// TwinCAT 3 PLC project ExternControl
// ProgramVersion: 3.1.4026.19
// libraries:
//   Tc2_Standard, * (Beckhoff Automation GmbH)
//   Tc2_System, * (Beckhoff Automation GmbH)
//   Tc2_Utilities, * (Beckhoff Automation GmbH)
//   VisuDialogs, * (System)
//   VisuDialogs
// project tree:
//   APPLICATION/ fb_Simulation.TcPOU, GVL_APPLICATION.TcGVL, MAIN_APP.TcPOU
//   APPLICATION/_types/ E_PROCESS_CHECK.TcDUT (not stored), E_PROCESS_CTRL.TcDUT (not stored), E_PROCESS_STATE.TcDUT (not stored), ST_PROCESS_CTRL.TcDUT (not stored), ST_PROCESS_STATE.TcDUT (not stored), T_PROCESS.TcDUT (not stored)
//   APPLICATION/_types/fb_Instance/ E_INSTANCE_CHECK.TcDUT, E_INSTANCE_STATE.TcDUT (not stored), fb_Instance.TcPOU (not stored)
//   APPLICATION/_types/LinkedList/ fb_Process_LinkedListCtrl.TcPOU (not stored), I_Process_LinkedList.TcIO (not stored), ST_PROCESS_DATA.TcDUT (not stored), ST_PROCESS_LIST_RESULT.TcDUT (not stored)
//   / GlobalTextList.TcGTLO (not stored), MAIN.TcPOU (not stored), PlcTask.TcTTO, Visualization Manager.TcVMO (not stored)
//   MAPPING/ MAPPING_in.TcPOU (not stored), MAPPING_out.TcPOU (not stored)
//   MAPPING/_types/ U_APP_CTRL.TcDUT (not stored), U_APP_STATE.TcDUT (not stored), U_INSTANCE_CTRL.TcDUT (not stored), U_INSTANCE_STATE.TcDUT (not stored), U_TICKET_LIST_CTRL.TcDUT (not stored), U_TICKET_LIST_DATA_INPUT.TcDUT (not stored), U_TICKET_LIST_DATA_OUTPUT.TcDUT (not stored), U_TICKET_LIST_STATE.TcDUT (not stored), U_XTS_STATION_CTRL.TcDUT (not stored), U_XTS_STATION_STATE.TcDUT (not stored), U_XTS_TRANSPORT_CTRL.TcDUT, U_XTS_TRANSPORT_STATE.TcDUT (not stored)
//   MSG/ fb_LocalTime.TcPOU (not stored), fb_MessageData.TcPOU (not stored), fb_MessageDataCtrl.TcPOU, f_MessageSet.TcPOU (not stored), GVL_MSG.TcGVL (not stored), I_MessageData.TcIO
//   MSG/types/ e_Device.TcDUT (not stored), E_MessageType.TcDUT (not stored), E_MESSAGE_BATCH.TcDUT (not stored), E_MESSAGE_CHECK.TcDUT (not stored), E_MESSAGE_CTRL.TcDUT (not stored), E_MESSAGE_FLOW.TcDUT (not stored), E_MESSAGE_STATE.TcDUT, e_Subdevice.TcDUT (not stored), ST_Message.TcDUT (not stored), ST_MESSAGE_CTRL.TcDUT (not stored), ST_MESSAGE_STATE.TcDUT (not stored), TL_E_MESSAGETYPE.TcTLO
//   XTS/CaGroup/types/ E_CA_GROUP_STATE.TcDUT (not stored), E_GROUP_CHECK.TcDUT (not stored), ST_GROUP_INFO.TcDUT
//   XTS/ GVL_XTS.TcGVL (not stored), XTS_Parameter.TcGVL (not stored)
//   XTS/Mover/types/ E_MOVER_CTRL.TcDUT (not stored), E_MOVER_STATE.TcDUT (not stored), ST_GEAR_DATA.TcDUT (not stored), ST_MOVER_CTRL.TcDUT (not stored), ST_MOVER_INFO.TcDUT, ST_MOVER_STATE.TcDUT (not stored), ST_MOVE_DATA.TcDUT (not stored)
//   XTS/Xpu/types/ E_XPU_CHECK.TcDUT (not stored), E_XPU_CTRL.TcDUT (not stored), E_XPU_INIT.TcDUT (not stored), E_XPU_STATE.TcDUT (not stored), ST_XPU_CTRL.TcDUT (not stored), ST_XPU_INFO.TcDUT, ST_XPU_STATE.TcDUT (not stored)
//   XTS/XtsStation/_types/ E_STATION_CTRL.TcDUT (not stored), E_STATION_GEAR_DISTANCE_AXIS.TcDUT (not stored), E_STATION_STATE.TcDUT (not stored), E_STATION_TYPE.TcDUT (not stored), ST_STATION_CTRL.TcDUT (not stored), ST_STATION_GEAR_PARAMETER.TcDUT (not stored), ST_STATION_LIST_RESULT.TcDUT (not stored), ST_STATION_MOVER_DATA.TcDUT (not stored), ST_STATION_PARAMETER.TcDUT, ST_STATION_STATE.TcDUT (not stored), T_NEST_OFFSET.TcDUT
//   XTS/XtsTransportUnit/types/ E_XTS_TRANSPORT_CHECK.TcDUT (not stored), E_XTS_TRANSPORT_CTRL.TcDUT (not stored), E_XTS_TRANSPORT_STATE.TcDUT (not stored), ST_XTS_TRANSPORT_CTRL.TcDUT (not stored), ST_XTS_TRANSPORT_STATE.TcDUT (not stored)
//   XTS/_types/ E_PROGRESS.TcDUT (not stored), f_GetProgress.TcPOU (not stored), f_GetState.TcPOU (not stored)
//   XTS/_Visualization/ GROUP_VISU.TcVIS (not stored), MOVER_VISU.TcVIS (not stored), STATION_VISU.TcVIS (not stored), XPU_VISU.TcVIS (not stored), XTS_TRANSPORT.TcVIS (not stored)
//   XTS/_Visualization/textlists/ TL_E_CTRL_MOVER.TcTLO (not stored), TL_E_CTRL_STATION.TcTLO (not stored), TL_E_CTRL_TRANSPORT.TcTLO (not stored), TL_E_CTRL_XPU.TcTLO (not stored)
//   XTS/_Visualization/types/ ST_XPU_STRINGS.TcDUT (not stored)
// real-time tasks:
//   TASK XTS Task 1: cycle T#250us, priority 1, ADS port 350
//   TASK XTS AUX Task 1: cycle T#250us, priority 2, ADS port 351
//   TASK XTS Task 2: cycle T#250us, priority 3, ADS port 352
//   TASK PlcTask: cycle T#2ms, priority 15, ADS port 353
//   TASK Job Task: cycle default, priority 32
// motion (NC):
//   TASK NC-Task 1: cycle T#2ms, priority 4, ADS port 501
//   TASK NC-Task 1 SVB: cycle T#10ms, priority 8, ADS port 511
//   AXIS Mover Axis 1 (id 1)
//     Dynamic: AccelerationMaximum=80000, DecelerationMaximum=80000, Acceleration=20000, Deceleration=20000, Jerk=200000
//     Velo: Maximum=4000
//     PositionAreaControl: Enable=false
//     TargetPosControl: Enable=false
//     OtherSettings: AllowMotionCmdToSlave=true, AllowMotionCmdToExtSetGenAxis=true
//     encoder EncType=28
//       EncPara: ModuloFactor=8000, ToleranceWndModuloStart=0.2, MaxCount=#xffffffff
//     drive DrvType=22
//       DrvPara: MaxCount=#xffffffff, DriveControlDWord=#x00000100
//         Analog: VeloReferenz=4200, TorqueSetpointScale=10
//         TimeComp: TaskDelayCycles=1
//     controller CtrType=1
//       CtrPara: PriorControlFactor=1
//         PosDiffControl: Range=10
//         Observer: BandWidth=20
//   AXIS Mover Axis 2 (id 2)
//     Dynamic: AccelerationMaximum=80000, DecelerationMaximum=80000, Acceleration=20000, Deceleration=20000, Jerk=200000
//     Velo: Maximum=4000
//     PositionAreaControl: Enable=false
//     TargetPosControl: Enable=false
//     OtherSettings: AllowMotionCmdToSlave=true, AllowMotionCmdToExtSetGenAxis=true
//     encoder EncType=28
//       EncPara: ModuloFactor=8000, ToleranceWndModuloStart=0.2, MaxCount=#xffffffff
//     drive DrvType=22
//       DrvPara: MaxCount=#xffffffff, DriveControlDWord=#x00000100
//         Analog: VeloReferenz=4200, TorqueSetpointScale=10
//         TimeComp: TaskDelayCycles=1
//     controller CtrType=1
//       CtrPara: PriorControlFactor=1
//         PosDiffControl: Range=10
//         Observer: BandWidth=20
//   AXIS Mover Axis 3 (id 3)
//     Dynamic: AccelerationMaximum=80000, DecelerationMaximum=80000, Acceleration=20000, Deceleration=20000, Jerk=200000
//     Velo: Maximum=4000
//     PositionAreaControl: Enable=false
//     TargetPosControl: Enable=false
//     OtherSettings: AllowMotionCmdToSlave=true, AllowMotionCmdToExtSetGenAxis=true
//     encoder EncType=28
//       EncPara: ModuloFactor=8000, ToleranceWndModuloStart=0.2, MaxCount=#xffffffff
//     drive DrvType=22
//       DrvPara: MaxCount=#xffffffff, DriveControlDWord=#x00000100
//         Analog: VeloReferenz=4200, TorqueSetpointScale=10
//         TimeComp: TaskDelayCycles=1
//     controller CtrType=1
//       CtrPara: PriorControlFactor=1
//         PosDiffControl: Range=10
//         Observer: BandWidth=20
//   AXIS Mover Axis 4 (id 4)
//     Dynamic: AccelerationMaximum=80000, DecelerationMaximum=80000, Acceleration=20000, Deceleration=20000, Jerk=200000
//     Velo: Maximum=4000
//     PositionAreaControl: Enable=false
//     TargetPosControl: Enable=false
//     OtherSettings: AllowMotionCmdToSlave=true, AllowMotionCmdToExtSetGenAxis=true
//     encoder EncType=28
//       EncPara: ModuloFactor=8000, ToleranceWndModuloStart=0.2, MaxCount=#xffffffff
//     drive DrvType=22
//       DrvPara: MaxCount=#xffffffff, DriveControlDWord=#x00000100
//         Analog: VeloReferenz=4200, TorqueSetpointScale=10
//         TimeComp: TaskDelayCycles=1
//     controller CtrType=1
//       CtrPara: PriorControlFactor=1
//         PosDiffControl: Range=10
//         Observer: BandWidth=20
//   AXIS Mover Axis 5 (id 5)
//     Dynamic: AccelerationMaximum=80000, DecelerationMaximum=80000, Acceleration=20000, Deceleration=20000, Jerk=200000
//     Velo: Maximum=4000
//     PositionAreaControl: Enable=false
//     TargetPosControl: Enable=false
//     OtherSettings: AllowMotionCmdToSlave=true, AllowMotionCmdToExtSetGenAxis=true
//     encoder EncType=28
//       EncPara: ModuloFactor=8000, ToleranceWndModuloStart=0.2, MaxCount=#xffffffff
//     drive DrvType=22
//       DrvPara: MaxCount=#xffffffff, DriveControlDWord=#x00000100
//         Analog: VeloReferenz=4200, TorqueSetpointScale=10
//         TimeComp: TaskDelayCycles=1
//     controller CtrType=1
//       CtrPara: PriorControlFactor=1
//         PosDiffControl: Range=10
//         Observer: BandWidth=20
//   AXIS Mover Axis 6 (id 6)
//     Dynamic: AccelerationMaximum=80000, DecelerationMaximum=80000, Acceleration=20000, Deceleration=20000, Jerk=200000
//     Velo: Maximum=4000
//     PositionAreaControl: Enable=false
//     TargetPosControl: Enable=false
//     OtherSettings: AllowMotionCmdToSlave=true, AllowMotionCmdToExtSetGenAxis=true
//     encoder EncType=28
//       EncPara: ModuloFactor=8000, ToleranceWndModuloStart=0.2, MaxCount=#xffffffff
//     drive DrvType=22
//       DrvPara: MaxCount=#xffffffff, DriveControlDWord=#x00000100
//         Analog: VeloReferenz=4200, TorqueSetpointScale=10
//         TimeComp: TaskDelayCycles=1
//     controller CtrType=1
//       CtrPara: PriorControlFactor=1
//         PosDiffControl: Range=10
//         Observer: BandWidth=20
//   AXIS Mover Axis 7 (id 7)
//     Dynamic: AccelerationMaximum=80000, DecelerationMaximum=80000, Acceleration=20000, Deceleration=20000, Jerk=200000
//     Velo: Maximum=4000
//     PositionAreaControl: Enable=false
//     TargetPosControl: Enable=false
//     OtherSettings: AllowMotionCmdToSlave=true, AllowMotionCmdToExtSetGenAxis=true
//     encoder EncType=28
//       EncPara: ModuloFactor=8000, ToleranceWndModuloStart=0.2, MaxCount=#xffffffff
//     drive DrvType=22
//       DrvPara: MaxCount=#xffffffff, DriveControlDWord=#x00000100
//         Analog: VeloReferenz=4200, TorqueSetpointScale=10
//         TimeComp: TaskDelayCycles=1
//     controller CtrType=1
//       CtrPara: PriorControlFactor=1
//         PosDiffControl: Range=10
//         Observer: BandWidth=20
//   AXIS Mover Axis 8 (id 8)
//     Dynamic: AccelerationMaximum=80000, DecelerationMaximum=80000, Acceleration=20000, Deceleration=20000, Jerk=200000
//     Velo: Maximum=4000
//     PositionAreaControl: Enable=false
//     TargetPosControl: Enable=false
//     OtherSettings: AllowMotionCmdToSlave=true, AllowMotionCmdToExtSetGenAxis=true
//     encoder EncType=28
//       EncPara: ModuloFactor=8000, ToleranceWndModuloStart=0.2, MaxCount=#xffffffff
//     drive DrvType=22
//       DrvPara: MaxCount=#xffffffff, DriveControlDWord=#x00000100
//         Analog: VeloReferenz=4200, TorqueSetpointScale=10
//         TimeComp: TaskDelayCycles=1
//     controller CtrType=1
//       CtrPara: PriorControlFactor=1
//         PosDiffControl: Range=10
//         Observer: BandWidth=20
//   AXIS Mover Axis 9 (id 9)
//     Dynamic: AccelerationMaximum=80000, DecelerationMaximum=80000, Acceleration=20000, Deceleration=20000, Jerk=200000
//     Velo: Maximum=4000
//     PositionAreaControl: Enable=false
//     TargetPosControl: Enable=false
//     OtherSettings: AllowMotionCmdToSlave=true, AllowMotionCmdToExtSetGenAxis=true
//     encoder EncType=28
//       EncPara: ModuloFactor=8000, ToleranceWndModuloStart=0.2, MaxCount=#xffffffff
//     drive DrvType=22
//       DrvPara: MaxCount=#xffffffff, DriveControlDWord=#x00000100
//         Analog: VeloReferenz=4200, TorqueSetpointScale=10
//         TimeComp: TaskDelayCycles=1
//     controller CtrType=1
//       CtrPara: PriorControlFactor=1
//         PosDiffControl: Range=10
//         Observer: BandWidth=20
//   AXIS Mover Axis 10 (id 10)
//     Dynamic: AccelerationMaximum=80000, DecelerationMaximum=80000, Acceleration=20000, Deceleration=20000, Jerk=200000
//     Velo: Maximum=4000
//     PositionAreaControl: Enable=false
//     TargetPosControl: Enable=false
//     OtherSettings: AllowMotionCmdToSlave=true, AllowMotionCmdToExtSetGenAxis=true
//     encoder EncType=28
//       EncPara: ModuloFactor=8000, ToleranceWndModuloStart=0.2, MaxCount=#xffffffff
//     drive DrvType=22
//       DrvPara: MaxCount=#xffffffff, DriveControlDWord=#x00000100
//         Analog: VeloReferenz=4200, TorqueSetpointScale=10
//         TimeComp: TaskDelayCycles=1
//     controller CtrType=1
//       CtrPara: PriorControlFactor=1
//         PosDiffControl: Range=10
//         Observer: BandWidth=20
//   AXIS Mover Axis 11 (id 11)
//     Dynamic: AccelerationMaximum=80000, DecelerationMaximum=80000, Acceleration=20000, Deceleration=20000, Jerk=200000
//     Velo: Maximum=4000
//     PositionAreaControl: Enable=false
//     TargetPosControl: Enable=false
//     OtherSettings: AllowMotionCmdToSlave=true, AllowMotionCmdToExtSetGenAxis=true
//     encoder EncType=28
//       EncPara: ModuloFactor=8000, ToleranceWndModuloStart=0.2, MaxCount=#xffffffff
//     drive DrvType=22
//       DrvPara: MaxCount=#xffffffff, DriveControlDWord=#x00000100
//         Analog: VeloReferenz=4200, TorqueSetpointScale=10
//         TimeComp: TaskDelayCycles=1
//     controller CtrType=1
//       CtrPara: PriorControlFactor=1
//         PosDiffControl: Range=10
//         Observer: BandWidth=20
//   AXIS Mover Axis 12 (id 12)
//     Dynamic: AccelerationMaximum=80000, DecelerationMaximum=80000, Acceleration=20000, Deceleration=20000, Jerk=200000
//     Velo: Maximum=4000
//     PositionAreaControl: Enable=false
//     TargetPosControl: Enable=false
//     OtherSettings: AllowMotionCmdToSlave=true, AllowMotionCmdToExtSetGenAxis=true
//     encoder EncType=28
//       EncPara: ModuloFactor=8000, ToleranceWndModuloStart=0.2, MaxCount=#xffffffff
//     drive DrvType=22
//       DrvPara: MaxCount=#xffffffff, DriveControlDWord=#x00000100
//         Analog: VeloReferenz=4200, TorqueSetpointScale=10
//         TimeComp: TaskDelayCycles=1
//     controller CtrType=1
//       CtrPara: PriorControlFactor=1
//         PosDiffControl: Range=10
//         Observer: BandWidth=20
//   AXIS Mover Axis 13 (id 13)
//     Dynamic: AccelerationMaximum=80000, DecelerationMaximum=80000, Acceleration=20000, Deceleration=20000, Jerk=200000
//     Velo: Maximum=4000
//     PositionAreaControl: Enable=false
//     TargetPosControl: Enable=false
//     OtherSettings: AllowMotionCmdToSlave=true, AllowMotionCmdToExtSetGenAxis=true
//     encoder EncType=28
//       EncPara: ModuloFactor=8000, ToleranceWndModuloStart=0.2, MaxCount=#xffffffff
//     drive DrvType=22
//       DrvPara: MaxCount=#xffffffff, DriveControlDWord=#x00000100
//         Analog: VeloReferenz=4200, TorqueSetpointScale=10
//         TimeComp: TaskDelayCycles=1
//     controller CtrType=1
//       CtrPara: PriorControlFactor=1
//         PosDiffControl: Range=10
//         Observer: BandWidth=20
//   AXIS Mover Axis 14 (id 14)
//     Dynamic: AccelerationMaximum=80000, DecelerationMaximum=80000, Acceleration=20000, Deceleration=20000, Jerk=200000
//     Velo: Maximum=4000
//     PositionAreaControl: Enable=false
//     TargetPosControl: Enable=false
//     OtherSettings: AllowMotionCmdToSlave=true, AllowMotionCmdToExtSetGenAxis=true
//     encoder EncType=28
//       EncPara: ModuloFactor=8000, ToleranceWndModuloStart=0.2, MaxCount=#xffffffff
//     drive DrvType=22
//       DrvPara: MaxCount=#xffffffff, DriveControlDWord=#x00000100
//         Analog: VeloReferenz=4200, TorqueSetpointScale=10
//         TimeComp: TaskDelayCycles=1
//     controller CtrType=1
//       CtrPara: PriorControlFactor=1
//         PosDiffControl: Range=10
//         Observer: BandWidth=20
//   AXIS Mover Axis 15 (id 15)
//     Dynamic: AccelerationMaximum=80000, DecelerationMaximum=80000, Acceleration=20000, Deceleration=20000, Jerk=200000
//     Velo: Maximum=4000
//     PositionAreaControl: Enable=false
//     TargetPosControl: Enable=false
//     OtherSettings: AllowMotionCmdToSlave=true, AllowMotionCmdToExtSetGenAxis=true
//     encoder EncType=28
//       EncPara: ModuloFactor=8000, ToleranceWndModuloStart=0.2, MaxCount=#xffffffff
//     drive DrvType=22
//       DrvPara: MaxCount=#xffffffff, DriveControlDWord=#x00000100
//         Analog: VeloReferenz=4200, TorqueSetpointScale=10
//         TimeComp: TaskDelayCycles=1
//     controller CtrType=1
//       CtrPara: PriorControlFactor=1
//         PosDiffControl: Range=10
//         Observer: BandWidth=20
//   AXIS Mover Axis 16 (id 16)
//     Dynamic: AccelerationMaximum=80000, DecelerationMaximum=80000, Acceleration=20000, Deceleration=20000, Jerk=200000
//     Velo: Maximum=4000
//     PositionAreaControl: Enable=false
//     TargetPosControl: Enable=false
//     OtherSettings: AllowMotionCmdToSlave=true, AllowMotionCmdToExtSetGenAxis=true
//     encoder EncType=28
//       EncPara: ModuloFactor=8000, ToleranceWndModuloStart=0.2, MaxCount=#xffffffff
//     drive DrvType=22
//       DrvPara: MaxCount=#xffffffff, DriveControlDWord=#x00000100
//         Analog: VeloReferenz=4200, TorqueSetpointScale=10
//         TimeComp: TaskDelayCycles=1
//     controller CtrType=1
//       CtrPara: PriorControlFactor=1
//         PosDiffControl: Range=10
//         Observer: BandWidth=20
//   AXIS Mover Axis 17 (id 17)
//     Dynamic: AccelerationMaximum=80000, DecelerationMaximum=80000, Acceleration=20000, Deceleration=20000, Jerk=200000
//     Velo: Maximum=4000
//     PositionAreaControl: Enable=false
//     TargetPosControl: Enable=false
//     OtherSettings: AllowMotionCmdToSlave=true, AllowMotionCmdToExtSetGenAxis=true
//     encoder EncType=28
//       EncPara: ModuloFactor=8000, ToleranceWndModuloStart=0.2, MaxCount=#xffffffff
//     drive DrvType=22
//       DrvPara: MaxCount=#xffffffff, DriveControlDWord=#x00000100
//         Analog: VeloReferenz=4200, TorqueSetpointScale=10
//         TimeComp: TaskDelayCycles=1
//     controller CtrType=1
//       CtrPara: PriorControlFactor=1
//         PosDiffControl: Range=10
//         Observer: BandWidth=20
//   AXIS Mover Axis 18 (id 18)
//     Dynamic: AccelerationMaximum=80000, DecelerationMaximum=80000, Acceleration=20000, Deceleration=20000, Jerk=200000
//     Velo: Maximum=4000
//     PositionAreaControl: Enable=false
//     TargetPosControl: Enable=false
//     OtherSettings: AllowMotionCmdToSlave=true, AllowMotionCmdToExtSetGenAxis=true
//     encoder EncType=28
//       EncPara: ModuloFactor=8000, ToleranceWndModuloStart=0.2, MaxCount=#xffffffff
//     drive DrvType=22
//       DrvPara: MaxCount=#xffffffff, DriveControlDWord=#x00000100
//         Analog: VeloReferenz=4200, TorqueSetpointScale=10
//         TimeComp: TaskDelayCycles=1
//     controller CtrType=1
//       CtrPara: PriorControlFactor=1
//         PosDiffControl: Range=10
//         Observer: BandWidth=20
//   AXIS Mover Axis 19 (id 19)
//     Dynamic: AccelerationMaximum=80000, DecelerationMaximum=80000, Acceleration=20000, Deceleration=20000, Jerk=200000
//     Velo: Maximum=4000
//     PositionAreaControl: Enable=false
//     TargetPosControl: Enable=false
//     OtherSettings: AllowMotionCmdToSlave=true, AllowMotionCmdToExtSetGenAxis=true
//     encoder EncType=28
//       EncPara: ModuloFactor=8000, ToleranceWndModuloStart=0.2, MaxCount=#xffffffff
//     drive DrvType=22
//       DrvPara: MaxCount=#xffffffff, DriveControlDWord=#x00000100
//         Analog: VeloReferenz=4200, TorqueSetpointScale=10
//         TimeComp: TaskDelayCycles=1
//     controller CtrType=1
//       CtrPara: PriorControlFactor=1
//         PosDiffControl: Range=10
//         Observer: BandWidth=20
//   AXIS Mover Axis 20 (id 20)
//     Dynamic: AccelerationMaximum=80000, DecelerationMaximum=80000, Acceleration=20000, Deceleration=20000, Jerk=200000
//     Velo: Maximum=4000
//     PositionAreaControl: Enable=false
//     TargetPosControl: Enable=false
//     OtherSettings: AllowMotionCmdToSlave=true, AllowMotionCmdToExtSetGenAxis=true
//     encoder EncType=28
//       EncPara: ModuloFactor=8000, ToleranceWndModuloStart=0.2, MaxCount=#xffffffff
//     drive DrvType=22
//       DrvPara: MaxCount=#xffffffff, DriveControlDWord=#x00000100
//         Analog: VeloReferenz=4200, TorqueSetpointScale=10
//         TimeComp: TaskDelayCycles=1
//     controller CtrType=1
//       CtrPara: PriorControlFactor=1
//         PosDiffControl: Range=10
//         Observer: BandWidth=20
//   AXIS Mover Axis 21 (id 21)
//     Dynamic: AccelerationMaximum=80000, DecelerationMaximum=80000, Acceleration=20000, Deceleration=20000, Jerk=200000
//     Velo: Maximum=4000
//     PositionAreaControl: Enable=false
//     TargetPosControl: Enable=false
//     OtherSettings: AllowMotionCmdToSlave=true, AllowMotionCmdToExtSetGenAxis=true
//     encoder EncType=28
//       EncPara: ModuloFactor=8000, ToleranceWndModuloStart=0.2, MaxCount=#xffffffff
//     drive DrvType=22
//       DrvPara: MaxCount=#xffffffff, DriveControlDWord=#x00000100
//         Analog: VeloReferenz=4200, TorqueSetpointScale=10
//         TimeComp: TaskDelayCycles=1
//     controller CtrType=1
//       CtrPara: PriorControlFactor=1
//         PosDiffControl: Range=10
//         Observer: BandWidth=20
//   AXIS Mover Axis 22 (id 22)
//     Dynamic: AccelerationMaximum=80000, DecelerationMaximum=80000, Acceleration=20000, Deceleration=20000, Jerk=200000
//     Velo: Maximum=4000
//     PositionAreaControl: Enable=false
//     TargetPosControl: Enable=false
//     OtherSettings: AllowMotionCmdToSlave=true, AllowMotionCmdToExtSetGenAxis=true
//     encoder EncType=28
//       EncPara: ModuloFactor=8000, ToleranceWndModuloStart=0.2, MaxCount=#xffffffff
//     drive DrvType=22
//       DrvPara: MaxCount=#xffffffff, DriveControlDWord=#x00000100
//         Analog: VeloReferenz=4200, TorqueSetpointScale=10
//         TimeComp: TaskDelayCycles=1
//     controller CtrType=1
//       CtrPara: PriorControlFactor=1
//         PosDiffControl: Range=10
//         Observer: BandWidth=20
//   AXIS Mover Axis 23 (id 23)
//     Dynamic: AccelerationMaximum=80000, DecelerationMaximum=80000, Acceleration=20000, Deceleration=20000, Jerk=200000
//     Velo: Maximum=4000
//     PositionAreaControl: Enable=false
//     TargetPosControl: Enable=false
//     OtherSettings: AllowMotionCmdToSlave=true, AllowMotionCmdToExtSetGenAxis=true
//     encoder EncType=28
//       EncPara: ModuloFactor=8000, ToleranceWndModuloStart=0.2, MaxCount=#xffffffff
//     drive DrvType=22
//       DrvPara: MaxCount=#xffffffff, DriveControlDWord=#x00000100
//         Analog: VeloReferenz=4200, TorqueSetpointScale=10
//         TimeComp: TaskDelayCycles=1
//     controller CtrType=1
//       CtrPara: PriorControlFactor=1
//         PosDiffControl: Range=10
//         Observer: BandWidth=20
//   AXIS Mover Axis 24 (id 24)
//     Dynamic: AccelerationMaximum=80000, DecelerationMaximum=80000, Acceleration=20000, Deceleration=20000, Jerk=200000
//     Velo: Maximum=4000
//     PositionAreaControl: Enable=false
//     TargetPosControl: Enable=false
//     OtherSettings: AllowMotionCmdToSlave=true, AllowMotionCmdToExtSetGenAxis=true
//     encoder EncType=28
//       EncPara: ModuloFactor=8000, ToleranceWndModuloStart=0.2, MaxCount=#xffffffff
//     drive DrvType=22
//       DrvPara: MaxCount=#xffffffff, DriveControlDWord=#x00000100
//         Analog: VeloReferenz=4200, TorqueSetpointScale=10
//         TimeComp: TaskDelayCycles=1
//     controller CtrType=1
//       CtrPara: PriorControlFactor=1
//         PosDiffControl: Range=10
//         Observer: BandWidth=20
//   AXIS Mover Axis 25 (id 25)
//     Dynamic: AccelerationMaximum=80000, DecelerationMaximum=80000, Acceleration=20000, Deceleration=20000, Jerk=200000
//     Velo: Maximum=4000
//     PositionAreaControl: Enable=false
//     TargetPosControl: Enable=false
//     OtherSettings: AllowMotionCmdToSlave=true, AllowMotionCmdToExtSetGenAxis=true
//     encoder EncType=28
//       EncPara: ModuloFactor=8000, ToleranceWndModuloStart=0.2, MaxCount=#xffffffff
//     drive DrvType=22
//       DrvPara: MaxCount=#xffffffff, DriveControlDWord=#x00000100
//         Analog: VeloReferenz=4200, TorqueSetpointScale=10
//         TimeComp: TaskDelayCycles=1
//     controller CtrType=1
//       CtrPara: PriorControlFactor=1
//         PosDiffControl: Range=10
//         Observer: BandWidth=20
//   AXIS Mover Axis 26 (id 26)
//     Dynamic: AccelerationMaximum=80000, DecelerationMaximum=80000, Acceleration=20000, Deceleration=20000, Jerk=200000
//     Velo: Maximum=4000
//     PositionAreaControl: Enable=false
//     TargetPosControl: Enable=false
//     OtherSettings: AllowMotionCmdToSlave=true, AllowMotionCmdToExtSetGenAxis=true
//     encoder EncType=28
//       EncPara: ModuloFactor=8000, ToleranceWndModuloStart=0.2, MaxCount=#xffffffff
//     drive DrvType=22
//       DrvPara: MaxCount=#xffffffff, DriveControlDWord=#x00000100
//         Analog: VeloReferenz=4200, TorqueSetpointScale=10
//         TimeComp: TaskDelayCycles=1
//     controller CtrType=1
//       CtrPara: PriorControlFactor=1
//         PosDiffControl: Range=10
//         Observer: BandWidth=20
//   AXIS Mover Axis 27 (id 27)
//     Dynamic: AccelerationMaximum=80000, DecelerationMaximum=80000, Acceleration=20000, Deceleration=20000, Jerk=200000
//     Velo: Maximum=4000
//     PositionAreaControl: Enable=false
//     TargetPosControl: Enable=false
//     OtherSettings: AllowMotionCmdToSlave=true, AllowMotionCmdToExtSetGenAxis=true
//     encoder EncType=28
//       EncPara: ModuloFactor=8000, ToleranceWndModuloStart=0.2, MaxCount=#xffffffff
//     drive DrvType=22
//       DrvPara: MaxCount=#xffffffff, DriveControlDWord=#x00000100
//         Analog: VeloReferenz=4200, TorqueSetpointScale=10
//         TimeComp: TaskDelayCycles=1
//     controller CtrType=1
//       CtrPara: PriorControlFactor=1
//         PosDiffControl: Range=10
//         Observer: BandWidth=20
//   AXIS Mover Axis 28 (id 28)
//     Dynamic: AccelerationMaximum=80000, DecelerationMaximum=80000, Acceleration=20000, Deceleration=20000, Jerk=200000
//     Velo: Maximum=4000
//     PositionAreaControl: Enable=false
//     TargetPosControl: Enable=false
//     OtherSettings: AllowMotionCmdToSlave=true, AllowMotionCmdToExtSetGenAxis=true
//     encoder EncType=28
//       EncPara: ModuloFactor=8000, ToleranceWndModuloStart=0.2, MaxCount=#xffffffff
//     drive DrvType=22
//       DrvPara: MaxCount=#xffffffff, DriveControlDWord=#x00000100
//         Analog: VeloReferenz=4200, TorqueSetpointScale=10
//         TimeComp: TaskDelayCycles=1
//     controller CtrType=1
//       CtrPara: PriorControlFactor=1
//         PosDiffControl: Range=10
//         Observer: BandWidth=20
//   AXIS Mover Axis 29 (id 29)
//     Dynamic: AccelerationMaximum=80000, DecelerationMaximum=80000, Acceleration=20000, Deceleration=20000, Jerk=200000
//     Velo: Maximum=4000
//     PositionAreaControl: Enable=false
//     TargetPosControl: Enable=false
//     OtherSettings: AllowMotionCmdToSlave=true, AllowMotionCmdToExtSetGenAxis=true
//     encoder EncType=28
//       EncPara: ModuloFactor=8000, ToleranceWndModuloStart=0.2, MaxCount=#xffffffff
//     drive DrvType=22
//       DrvPara: MaxCount=#xffffffff, DriveControlDWord=#x00000100
//         Analog: VeloReferenz=4200, TorqueSetpointScale=10
//         TimeComp: TaskDelayCycles=1
//     controller CtrType=1
//       CtrPara: PriorControlFactor=1
//         PosDiffControl: Range=10
//         Observer: BandWidth=20
//   AXIS Mover Axis 30 (id 30)
//     Dynamic: AccelerationMaximum=80000, DecelerationMaximum=80000, Acceleration=20000, Deceleration=20000, Jerk=200000
//     Velo: Maximum=4000
//     PositionAreaControl: Enable=false
//     TargetPosControl: Enable=false
//     OtherSettings: AllowMotionCmdToSlave=true, AllowMotionCmdToExtSetGenAxis=true
//     encoder EncType=28
//       EncPara: ModuloFactor=8000, ToleranceWndModuloStart=0.2, MaxCount=#xffffffff
//     drive DrvType=22
//       DrvPara: MaxCount=#xffffffff, DriveControlDWord=#x00000100
//         Analog: VeloReferenz=4200, TorqueSetpointScale=10
//         TimeComp: TaskDelayCycles=1
//     controller CtrType=1
//       CtrPara: PriorControlFactor=1
//         PosDiffControl: Range=10
//         Observer: BandWidth=20
//   AXIS Mover Axis 31 (id 31)
//     Dynamic: AccelerationMaximum=80000, DecelerationMaximum=80000, Acceleration=20000, Deceleration=20000, Jerk=200000
//     Velo: Maximum=4000
//     PositionAreaControl: Enable=false
//     TargetPosControl: Enable=false
//     OtherSettings: AllowMotionCmdToSlave=true, AllowMotionCmdToExtSetGenAxis=true
//     encoder EncType=28
//       EncPara: ModuloFactor=8000, ToleranceWndModuloStart=0.2, MaxCount=#xffffffff
//     drive DrvType=22
//       DrvPara: MaxCount=#xffffffff, DriveControlDWord=#x00000100
//         Analog: VeloReferenz=4200, TorqueSetpointScale=10
//         TimeComp: TaskDelayCycles=1
//     controller CtrType=1
//       CtrPara: PriorControlFactor=1
//         PosDiffControl: Range=10
//         Observer: BandWidth=20
//   AXIS Mover Axis 32 (id 32)
//     Dynamic: AccelerationMaximum=80000, DecelerationMaximum=80000, Acceleration=20000, Deceleration=20000, Jerk=200000
//     Velo: Maximum=4000
//     PositionAreaControl: Enable=false
//     TargetPosControl: Enable=false
//     OtherSettings: AllowMotionCmdToSlave=true, AllowMotionCmdToExtSetGenAxis=true
//     encoder EncType=28
//       EncPara: ModuloFactor=8000, ToleranceWndModuloStart=0.2, MaxCount=#xffffffff
//     drive DrvType=22
//       DrvPara: MaxCount=#xffffffff, DriveControlDWord=#x00000100
//         Analog: VeloReferenz=4200, TorqueSetpointScale=10
//         TimeComp: TaskDelayCycles=1
//     controller CtrType=1
//       CtrPara: PriorControlFactor=1
//         PosDiffControl: Range=10
//         Observer: BandWidth=20
//   AXIS Mover Axis 33 (id 33)
//     Dynamic: AccelerationMaximum=80000, DecelerationMaximum=80000, Acceleration=20000, Deceleration=20000, Jerk=200000
//     Velo: Maximum=4000
//     PositionAreaControl: Enable=false
//     TargetPosControl: Enable=false
//     OtherSettings: AllowMotionCmdToSlave=true, AllowMotionCmdToExtSetGenAxis=true
//     encoder EncType=28
//       EncPara: ModuloFactor=8000, ToleranceWndModuloStart=0.2, MaxCount=#xffffffff
//     drive DrvType=22
//       DrvPara: MaxCount=#xffffffff, DriveControlDWord=#x00000100
//         Analog: VeloReferenz=4200, TorqueSetpointScale=10
//         TimeComp: TaskDelayCycles=1
//     controller CtrType=1
//       CtrPara: PriorControlFactor=1
//         PosDiffControl: Range=10
//         Observer: BandWidth=20
//   AXIS Mover Axis 34 (id 34)
//     Dynamic: AccelerationMaximum=80000, DecelerationMaximum=80000, Acceleration=20000, Deceleration=20000, Jerk=200000
//     Velo: Maximum=4000
//     PositionAreaControl: Enable=false
//     TargetPosControl: Enable=false
//     OtherSettings: AllowMotionCmdToSlave=true, AllowMotionCmdToExtSetGenAxis=true
//     encoder EncType=28
//       EncPara: ModuloFactor=8000, ToleranceWndModuloStart=0.2, MaxCount=#xffffffff
//     drive DrvType=22
//       DrvPara: MaxCount=#xffffffff, DriveControlDWord=#x00000100
//         Analog: VeloReferenz=4200, TorqueSetpointScale=10
//         TimeComp: TaskDelayCycles=1
//     controller CtrType=1
//       CtrPara: PriorControlFactor=1
//         PosDiffControl: Range=10
//         Observer: BandWidth=20
//   AXIS Mover Axis 35 (id 35)
//     Dynamic: AccelerationMaximum=80000, DecelerationMaximum=80000, Acceleration=20000, Deceleration=20000, Jerk=200000
//     Velo: Maximum=4000
//     PositionAreaControl: Enable=false
//     TargetPosControl: Enable=false
//     OtherSettings: AllowMotionCmdToSlave=true, AllowMotionCmdToExtSetGenAxis=true
//     encoder EncType=28
//       EncPara: ModuloFactor=8000, ToleranceWndModuloStart=0.2, MaxCount=#xffffffff
//     drive DrvType=22
//       DrvPara: MaxCount=#xffffffff, DriveControlDWord=#x00000100
//         Analog: VeloReferenz=4200, TorqueSetpointScale=10
//         TimeComp: TaskDelayCycles=1
//     controller CtrType=1
//       CtrPara: PriorControlFactor=1
//         PosDiffControl: Range=10
//         Observer: BandWidth=20
//   AXIS Mover Axis 36 (id 36)
//     Dynamic: AccelerationMaximum=80000, DecelerationMaximum=80000, Acceleration=20000, Deceleration=20000, Jerk=200000
//     Velo: Maximum=4000
//     PositionAreaControl: Enable=false
//     TargetPosControl: Enable=false
//     OtherSettings: AllowMotionCmdToSlave=true, AllowMotionCmdToExtSetGenAxis=true
//     encoder EncType=28
//       EncPara: ModuloFactor=8000, ToleranceWndModuloStart=0.2, MaxCount=#xffffffff
//     drive DrvType=22
//       DrvPara: MaxCount=#xffffffff, DriveControlDWord=#x00000100
//         Analog: VeloReferenz=4200, TorqueSetpointScale=10
//         TimeComp: TaskDelayCycles=1
//     controller CtrType=1
//       CtrPara: PriorControlFactor=1
//         PosDiffControl: Range=10
//         Observer: BandWidth=20
//   AXIS Mover Axis 37 (id 37)
//     Dynamic: AccelerationMaximum=80000, DecelerationMaximum=80000, Acceleration=20000, Deceleration=20000, Jerk=200000
//     Velo: Maximum=4000
//     PositionAreaControl: Enable=false
//     TargetPosControl: Enable=false
//     OtherSettings: AllowMotionCmdToSlave=true, AllowMotionCmdToExtSetGenAxis=true
//     encoder EncType=28
//       EncPara: ModuloFactor=8000, ToleranceWndModuloStart=0.2, MaxCount=#xffffffff
//     drive DrvType=22
//       DrvPara: MaxCount=#xffffffff, DriveControlDWord=#x00000100
//         Analog: VeloReferenz=4200, TorqueSetpointScale=10
//         TimeComp: TaskDelayCycles=1
//     controller CtrType=1
//       CtrPara: PriorControlFactor=1
//         PosDiffControl: Range=10
//         Observer: BandWidth=20
//   AXIS Mover Axis 38 (id 38)
//     Dynamic: AccelerationMaximum=80000, DecelerationMaximum=80000, Acceleration=20000, Deceleration=20000, Jerk=200000
//     Velo: Maximum=4000
//     PositionAreaControl: Enable=false
//     TargetPosControl: Enable=false
//     OtherSettings: AllowMotionCmdToSlave=true, AllowMotionCmdToExtSetGenAxis=true
//     encoder EncType=28
//       EncPara: ModuloFactor=8000, ToleranceWndModuloStart=0.2, MaxCount=#xffffffff
//     drive DrvType=22
//       DrvPara: MaxCount=#xffffffff, DriveControlDWord=#x00000100
//         Analog: VeloReferenz=4200, TorqueSetpointScale=10
//         TimeComp: TaskDelayCycles=1
//     controller CtrType=1
//       CtrPara: PriorControlFactor=1
//         PosDiffControl: Range=10
//         Observer: BandWidth=20
//   AXIS Mover Axis 39 (id 39)
//     Dynamic: AccelerationMaximum=80000, DecelerationMaximum=80000, Acceleration=20000, Deceleration=20000, Jerk=200000
//     Velo: Maximum=4000
//     PositionAreaControl: Enable=false
//     TargetPosControl: Enable=false
//     OtherSettings: AllowMotionCmdToSlave=true, AllowMotionCmdToExtSetGenAxis=true
//     encoder EncType=28
//       EncPara: ModuloFactor=8000, ToleranceWndModuloStart=0.2, MaxCount=#xffffffff
//     drive DrvType=22
//       DrvPara: MaxCount=#xffffffff, DriveControlDWord=#x00000100
//         Analog: VeloReferenz=4200, TorqueSetpointScale=10
//         TimeComp: TaskDelayCycles=1
//     controller CtrType=1
//       CtrPara: PriorControlFactor=1
//         PosDiffControl: Range=10
//         Observer: BandWidth=20
//   AXIS Mover Axis 40 (id 40)
//     Dynamic: AccelerationMaximum=80000, DecelerationMaximum=80000, Acceleration=20000, Deceleration=20000, Jerk=200000
//     Velo: Maximum=4000
//     PositionAreaControl: Enable=false
//     TargetPosControl: Enable=false
//     OtherSettings: AllowMotionCmdToSlave=true, AllowMotionCmdToExtSetGenAxis=true
//     encoder EncType=28
//       EncPara: ModuloFactor=8000, ToleranceWndModuloStart=0.2, MaxCount=#xffffffff
//     drive DrvType=22
//       DrvPara: MaxCount=#xffffffff, DriveControlDWord=#x00000100
//         Analog: VeloReferenz=4200, TorqueSetpointScale=10
//         TimeComp: TaskDelayCycles=1
//     controller CtrType=1
//       CtrPara: PriorControlFactor=1
//         PosDiffControl: Range=10
//         Observer: BandWidth=20
//   AXIS Mover Axis 41 (id 41)
//     Dynamic: AccelerationMaximum=80000, DecelerationMaximum=80000, Acceleration=20000, Deceleration=20000, Jerk=200000
//     Velo: Maximum=4000
//     PositionAreaControl: Enable=false
//     TargetPosControl: Enable=false
//     OtherSettings: AllowMotionCmdToSlave=true, AllowMotionCmdToExtSetGenAxis=true
//     encoder EncType=28
//       EncPara: ModuloFactor=8000, ToleranceWndModuloStart=0.2, MaxCount=#xffffffff
//     drive DrvType=22
//       DrvPara: MaxCount=#xffffffff, DriveControlDWord=#x00000100
//         Analog: VeloReferenz=4200, TorqueSetpointScale=10
//         TimeComp: TaskDelayCycles=1
//     controller CtrType=1
//       CtrPara: PriorControlFactor=1
//         PosDiffControl: Range=10
//         Observer: BandWidth=20
//   AXIS Mover Axis 42 (id 42)
//     Dynamic: AccelerationMaximum=80000, DecelerationMaximum=80000, Acceleration=20000, Deceleration=20000, Jerk=200000
//     Velo: Maximum=4000
//     PositionAreaControl: Enable=false
//     TargetPosControl: Enable=false
//     OtherSettings: AllowMotionCmdToSlave=true, AllowMotionCmdToExtSetGenAxis=true
//     encoder EncType=28
//       EncPara: ModuloFactor=8000, ToleranceWndModuloStart=0.2, MaxCount=#xffffffff
//     drive DrvType=22
//       DrvPara: MaxCount=#xffffffff, DriveControlDWord=#x00000100
//         Analog: VeloReferenz=4200, TorqueSetpointScale=10
//         TimeComp: TaskDelayCycles=1
//     controller CtrType=1
//       CtrPara: PriorControlFactor=1
//         PosDiffControl: Range=10
//         Observer: BandWidth=20
//   AXIS Mover Axis 43 (id 43)
//     Dynamic: AccelerationMaximum=80000, DecelerationMaximum=80000, Acceleration=20000, Deceleration=20000, Jerk=200000
//     Velo: Maximum=4000
//     PositionAreaControl: Enable=false
//     TargetPosControl: Enable=false
//     OtherSettings: AllowMotionCmdToSlave=true, AllowMotionCmdToExtSetGenAxis=true
//     encoder EncType=28
//       EncPara: ModuloFactor=8000, ToleranceWndModuloStart=0.2, MaxCount=#xffffffff
//     drive DrvType=22
//       DrvPara: MaxCount=#xffffffff, DriveControlDWord=#x00000100
//         Analog: VeloReferenz=4200, TorqueSetpointScale=10
//         TimeComp: TaskDelayCycles=1
//     controller CtrType=1
//       CtrPara: PriorControlFactor=1
//         PosDiffControl: Range=10
//         Observer: BandWidth=20
//   AXIS Mover Axis 44 (id 44)
//     Dynamic: AccelerationMaximum=80000, DecelerationMaximum=80000, Acceleration=20000, Deceleration=20000, Jerk=200000
//     Velo: Maximum=4000
//     PositionAreaControl: Enable=false
//     TargetPosControl: Enable=false
//     OtherSettings: AllowMotionCmdToSlave=true, AllowMotionCmdToExtSetGenAxis=true
//     encoder EncType=28
//       EncPara: ModuloFactor=8000, ToleranceWndModuloStart=0.2, MaxCount=#xffffffff
//     drive DrvType=22
//       DrvPara: MaxCount=#xffffffff, DriveControlDWord=#x00000100
//         Analog: VeloReferenz=4200, TorqueSetpointScale=10
//         TimeComp: TaskDelayCycles=1
//     controller CtrType=1
//       CtrPara: PriorControlFactor=1
//         PosDiffControl: Range=10
//         Observer: BandWidth=20
//   AXIS Mover Axis 45 (id 45)
//     Dynamic: AccelerationMaximum=80000, DecelerationMaximum=80000, Acceleration=20000, Deceleration=20000, Jerk=200000
//     Velo: Maximum=4000
//     PositionAreaControl: Enable=false
//     TargetPosControl: Enable=false
//     OtherSettings: AllowMotionCmdToSlave=true, AllowMotionCmdToExtSetGenAxis=true
//     encoder EncType=28
//       EncPara: ModuloFactor=8000, ToleranceWndModuloStart=0.2, MaxCount=#xffffffff
//     drive DrvType=22
//       DrvPara: MaxCount=#xffffffff, DriveControlDWord=#x00000100
//         Analog: VeloReferenz=4200, TorqueSetpointScale=10
//         TimeComp: TaskDelayCycles=1
//     controller CtrType=1
//       CtrPara: PriorControlFactor=1
//         PosDiffControl: Range=10
//         Observer: BandWidth=20
//   AXIS Mover Axis 46 (id 46)
//     Dynamic: AccelerationMaximum=80000, DecelerationMaximum=80000, Acceleration=20000, Deceleration=20000, Jerk=200000
//     Velo: Maximum=4000
//     PositionAreaControl: Enable=false
//     TargetPosControl: Enable=false
//     OtherSettings: AllowMotionCmdToSlave=true, AllowMotionCmdToExtSetGenAxis=true
//     encoder EncType=28
//       EncPara: ModuloFactor=8000, ToleranceWndModuloStart=0.2, MaxCount=#xffffffff
//     drive DrvType=22
//       DrvPara: MaxCount=#xffffffff, DriveControlDWord=#x00000100
//         Analog: VeloReferenz=4200, TorqueSetpointScale=10
//         TimeComp: TaskDelayCycles=1
//     controller CtrType=1
//       CtrPara: PriorControlFactor=1
//         PosDiffControl: Range=10
//         Observer: BandWidth=20
//   AXIS Mover Axis 47 (id 47)
//     Dynamic: AccelerationMaximum=80000, DecelerationMaximum=80000, Acceleration=20000, Deceleration=20000, Jerk=200000
//     Velo: Maximum=4000
//     PositionAreaControl: Enable=false
//     TargetPosControl: Enable=false
//     OtherSettings: AllowMotionCmdToSlave=true, AllowMotionCmdToExtSetGenAxis=true
//     encoder EncType=28
//       EncPara: ModuloFactor=8000, ToleranceWndModuloStart=0.2, MaxCount=#xffffffff
//     drive DrvType=22
//       DrvPara: MaxCount=#xffffffff, DriveControlDWord=#x00000100
//         Analog: VeloReferenz=4200, TorqueSetpointScale=10
//         TimeComp: TaskDelayCycles=1
//     controller CtrType=1
//       CtrPara: PriorControlFactor=1
//         PosDiffControl: Range=10
//         Observer: BandWidth=20
//   AXIS Mover Axis 48 (id 48)
//     Dynamic: AccelerationMaximum=80000, DecelerationMaximum=80000, Acceleration=20000, Deceleration=20000, Jerk=200000
//     Velo: Maximum=4000
//     PositionAreaControl: Enable=false
//     TargetPosControl: Enable=false
//     OtherSettings: AllowMotionCmdToSlave=true, AllowMotionCmdToExtSetGenAxis=true
//     encoder EncType=28
//       EncPara: ModuloFactor=8000, ToleranceWndModuloStart=0.2, MaxCount=#xffffffff
//     drive DrvType=22
//       DrvPara: MaxCount=#xffffffff, DriveControlDWord=#x00000100
//         Analog: VeloReferenz=4200, TorqueSetpointScale=10
//         TimeComp: TaskDelayCycles=1
//     controller CtrType=1
//       CtrPara: PriorControlFactor=1
//         PosDiffControl: Range=10
//         Observer: BandWidth=20
// I/O:
//   DEVICE Device 1 (disabled), AmsNetId 5.163.199.237.2.1
//     Term 1 (AT2002-0250) [AT2002-0250 Motor module with feed (B23-Connector) 250 mm, 48V]
//       Term 2 (AT2002-5250) [AT2002-5250 Sensor line with feed (B23-Connector)]
//     Term 3 (AT2000-0250) [AT2000-0250 Motor module 250 mm, 48V]
//       Term 4 (AT2000-5250) [AT2000-5250 Sensor line]
//     Term 5 (AT2000-0250) [AT2000-0250 Motor module 250 mm, 48V]
//       Term 6 (AT2000-5250) [AT2000-5250 Sensor line]
//     Term 7 (AT2000-0250) [AT2000-0250 Motor module 250 mm, 48V]
//       Term 8 (AT2000-5250) [AT2000-5250 Sensor line]
//   DEVICE Device 3 (disabled), AmsNetId 5.163.199.237.3.1
//     Term 9 (AT2002-0250) [AT2002-0250 Motor module with feed (B23-Connector) 250 mm, 48V]
//       Term 10 (AT2002-5250) [AT2002-5250 Sensor line with feed (B23-Connector)]
//     Term 11 (AT2000-0250) [AT2000-0250 Motor module 250 mm, 48V]
//       Term 12 (AT2000-5250) [AT2000-5250 Sensor line]
//     Term 13 (AT2000-0250) [AT2000-0250 Motor module 250 mm, 48V]
//       Term 14 (AT2000-5250) [AT2000-5250 Sensor line]
//     Term 15 (AT2000-0250) [AT2000-0250 Motor module 250 mm, 48V]
//       Term 16 (AT2000-5250) [AT2000-5250 Sensor line]
//   DEVICE Device 4 (disabled), AmsNetId 5.163.199.237.4.1
//     Term 17 (AT2002-0250) [AT2002-0250 Motor module with feed (B23-Connector) 250 mm, 48V]
//       Term 18 (AT2002-5250) [AT2002-5250 Sensor line with feed (B23-Connector)]
//     Term 19 (AT2040-0250) [AT2040-0250 Motor module, +45°, 250mm, 48V]
//       Term 20 (AT2040-5250) [AT2040-5250 Sensor line +45°]
//     Term 21 (AT2040-0250) [AT2040-0250 Motor module, +45°, 250mm, 48V]
//       Term 22 (AT2040-5250) [AT2040-5250 Sensor line +45°]
//     Term 23 (AT2000-0250) [AT2000-0250 Motor module 250 mm, 48V]
//       Term 24 (AT2000-5250) [AT2000-5250 Sensor line]
//   DEVICE Device 5 (disabled), AmsNetId 5.163.199.237.5.1
//     Term 25 (AT2002-0250) [AT2002-0250 Motor module with feed (B23-Connector) 250 mm, 48V]
//       Term 26 (AT2002-5250) [AT2002-5250 Sensor line with feed (B23-Connector)]
//     Term 27 (AT2000-0250) [AT2000-0250 Motor module 250 mm, 48V]
//       Term 28 (AT2000-5250) [AT2000-5250 Sensor line]
//     Term 29 (AT2040-0250) [AT2040-0250 Motor module, +45°, 250mm, 48V]
//       Term 30 (AT2040-5250) [AT2040-5250 Sensor line +45°]
//     Term 31 (AT2040-0250) [AT2040-0250 Motor module, +45°, 250mm, 48V]
//       Term 32 (AT2040-5250) [AT2040-5250 Sensor line +45°]
//     Term 33 (AT2000-0250) [AT2000-0250 Motor module 250 mm, 48V]
//       Term 34 (AT2000-5250) [AT2000-5250 Sensor line]
//   DEVICE Device 6 (disabled), AmsNetId 5.163.199.237.6.1
//     Term 35 (AT2002-0250) [AT2002-0250 Motor module with feed (B23-Connector) 250 mm, 48V]
//       Term 36 (AT2002-5250) [AT2002-5250 Sensor line with feed (B23-Connector)]
//     Term 37 (AT2000-0250) [AT2000-0250 Motor module 250 mm, 48V]
//       Term 38 (AT2000-5250) [AT2000-5250 Sensor line]
//     Term 39 (AT2000-0250) [AT2000-0250 Motor module 250 mm, 48V]
//       Term 40 (AT2000-5250) [AT2000-5250 Sensor line]
//     Term 41 (AT2000-0250) [AT2000-0250 Motor module 250 mm, 48V]
//       Term 42 (AT2000-5250) [AT2000-5250 Sensor line]
//   DEVICE Device 7 (disabled), AmsNetId 5.163.199.237.7.1
//     Term 43 (AT2002-0250) [AT2002-0250 Motor module with feed (B23-Connector) 250 mm, 48V]
//       Term 44 (AT2002-5250) [AT2002-5250 Sensor line with feed (B23-Connector)]
//     Term 45 (AT2000-0250) [AT2000-0250 Motor module 250 mm, 48V]
//       Term 46 (AT2000-5250) [AT2000-5250 Sensor line]
//     Term 47 (AT2000-0250) [AT2000-0250 Motor module 250 mm, 48V]
//       Term 48 (AT2000-5250) [AT2000-5250 Sensor line]
//     Term 49 (AT2000-0250) [AT2000-0250 Motor module 250 mm, 48V]
//       Term 50 (AT2000-5250) [AT2000-5250 Sensor line]
//   DEVICE Device 8 (disabled), AmsNetId 5.163.199.237.8.1
//     Term 51 (AT2042-0250) [AT2042-0250 Motor module with feed (B23-Connector), +45°, 250 mm, 48V]
//       Term 52 (AT2042-5250) [AT2042-5250 Sensor line with feed (B23-Connector), +45°]
//     Term 53 (AT2040-0250) [AT2040-0250 Motor module, +45°, 250mm, 48V]
//       Term 54 (AT2040-5250) [AT2040-5250 Sensor line +45°]
//     Term 55 (AT2000-0250) [AT2000-0250 Motor module 250 mm, 48V]
//       Term 56 (AT2000-5250) [AT2000-5250 Sensor line]
//     Term 57 (AT2000-0250) [AT2000-0250 Motor module 250 mm, 48V]
//       Term 58 (AT2000-5250) [AT2000-5250 Sensor line]
//   DEVICE Device 9 (disabled), AmsNetId 5.163.199.237.9.1
//     Term 59 (AT2002-0250) [AT2002-0250 Motor module with feed (B23-Connector) 250 mm, 48V]
//       Term 60 (AT2002-5250) [AT2002-5250 Sensor line with feed (B23-Connector)]
//     Term 61 (AT2040-0250) [AT2040-0250 Motor module, +45°, 250mm, 48V]
//       Term 62 (AT2040-5250) [AT2040-5250 Sensor line +45°]
//     Term 63 (AT2040-0250) [AT2040-0250 Motor module, +45°, 250mm, 48V]
//       Term 64 (AT2040-5250) [AT2040-5250 Sensor line +45°]
// variable links:
//   Device 1 <-> TcCOM Objects/XTS ProcessingUnit 1/Part 1/Module 1
//     Term 1 (AT2002-0250)/CC Inputs/Current actual value Ch.1 <-> Data Pointer/CurrentActualValues[0]
//     Term 1 (AT2002-0250)/CC Inputs/Current actual value Ch.10 <-> Data Pointer/CurrentActualValues[9]
//     Term 1 (AT2002-0250)/CC Inputs/Current actual value Ch.11 <-> Data Pointer/CurrentActualValues[10]
//     Term 1 (AT2002-0250)/CC Inputs/Current actual value Ch.12 <-> Data Pointer/CurrentActualValues[11]
//     Term 1 (AT2002-0250)/CC Inputs/Current actual value Ch.13 <-> Data Pointer/CurrentActualValues[12]
//     Term 1 (AT2002-0250)/CC Inputs/Current actual value Ch.14 <-> Data Pointer/CurrentActualValues[13]
//     Term 1 (AT2002-0250)/CC Inputs/Current actual value Ch.15 <-> Data Pointer/CurrentActualValues[14]
//     Term 1 (AT2002-0250)/CC Inputs/Current actual value Ch.2 <-> Data Pointer/CurrentActualValues[1]
//     Term 1 (AT2002-0250)/CC Inputs/Current actual value Ch.3 <-> Data Pointer/CurrentActualValues[2]
//     Term 1 (AT2002-0250)/CC Inputs/Current actual value Ch.4 <-> Data Pointer/CurrentActualValues[3]
//     Term 1 (AT2002-0250)/CC Inputs/Current actual value Ch.5 <-> Data Pointer/CurrentActualValues[4]
//     Term 1 (AT2002-0250)/CC Inputs/Current actual value Ch.6 <-> Data Pointer/CurrentActualValues[5]
//     Term 1 (AT2002-0250)/CC Inputs/Current actual value Ch.7 <-> Data Pointer/CurrentActualValues[6]
//     Term 1 (AT2002-0250)/CC Inputs/Current actual value Ch.8 <-> Data Pointer/CurrentActualValues[7]
//     Term 1 (AT2002-0250)/CC Inputs/Current actual value Ch.9 <-> Data Pointer/CurrentActualValues[8]
//     Term 1 (AT2002-0250)/CC Inputs/Status <-> Data Pointer/Status
//     Term 1 (AT2002-0250)/CC Outputs/Control <-> Data Pointer/Control
//     Term 1 (AT2002-0250)/CC Outputs/Current setpoint value Ch.1 <-> Data Pointer/CurrentSetpointValues[0]
//     Term 1 (AT2002-0250)/CC Outputs/Current setpoint value Ch.10 <-> Data Pointer/CurrentSetpointValues[9]
//     Term 1 (AT2002-0250)/CC Outputs/Current setpoint value Ch.11 <-> Data Pointer/CurrentSetpointValues[10]
//     Term 1 (AT2002-0250)/CC Outputs/Current setpoint value Ch.12 <-> Data Pointer/CurrentSetpointValues[11]
//     Term 1 (AT2002-0250)/CC Outputs/Current setpoint value Ch.13 <-> Data Pointer/CurrentSetpointValues[12]
//     Term 1 (AT2002-0250)/CC Outputs/Current setpoint value Ch.14 <-> Data Pointer/CurrentSetpointValues[13]
//     Term 1 (AT2002-0250)/CC Outputs/Current setpoint value Ch.15 <-> Data Pointer/CurrentSetpointValues[14]
//     Term 1 (AT2002-0250)/CC Outputs/Current setpoint value Ch.2 <-> Data Pointer/CurrentSetpointValues[1]
//     Term 1 (AT2002-0250)/CC Outputs/Current setpoint value Ch.3 <-> Data Pointer/CurrentSetpointValues[2]
//     Term 1 (AT2002-0250)/CC Outputs/Current setpoint value Ch.4 <-> Data Pointer/CurrentSetpointValues[3]
//     Term 1 (AT2002-0250)/CC Outputs/Current setpoint value Ch.5 <-> Data Pointer/CurrentSetpointValues[4]
//     Term 1 (AT2002-0250)/CC Outputs/Current setpoint value Ch.6 <-> Data Pointer/CurrentSetpointValues[5]
//     Term 1 (AT2002-0250)/CC Outputs/Current setpoint value Ch.7 <-> Data Pointer/CurrentSetpointValues[6]
//     Term 1 (AT2002-0250)/CC Outputs/Current setpoint value Ch.8 <-> Data Pointer/CurrentSetpointValues[7]
//     Term 1 (AT2002-0250)/CC Outputs/Current setpoint value Ch.9 <-> Data Pointer/CurrentSetpointValues[8]
//     Term 1 (AT2002-0250)/Term 2 (AT2002-5250)/FB Inputs/Value Channel 01 <-> Data Pointer/RawPositionValues[0]
//     Term 1 (AT2002-0250)/Term 2 (AT2002-5250)/FB Inputs/Value Channel 02 <-> Data Pointer/RawPositionValues[1]
//     Term 1 (AT2002-0250)/Term 2 (AT2002-5250)/FB Inputs/Value Channel 03 <-> Data Pointer/RawPositionValues[2]
//     Term 1 (AT2002-0250)/Term 2 (AT2002-5250)/FB Inputs/Value Channel 04 <-> Data Pointer/RawPositionValues[3]
//     Term 1 (AT2002-0250)/Term 2 (AT2002-5250)/FB Inputs/Value Channel 05 <-> Data Pointer/RawPositionValues[4]
//     Term 1 (AT2002-0250)/Term 2 (AT2002-5250)/FB Inputs/Value Channel 06 <-> Data Pointer/RawPositionValues[5]
//     Term 1 (AT2002-0250)/Term 2 (AT2002-5250)/FB Inputs/Value Channel 07 <-> Data Pointer/RawPositionValues[6]
//     Term 1 (AT2002-0250)/Term 2 (AT2002-5250)/FB Inputs/Value Channel 08 <-> Data Pointer/RawPositionValues[7]
//     Term 1 (AT2002-0250)/Term 2 (AT2002-5250)/FB Inputs/Value Channel 09 <-> Data Pointer/RawPositionValues[8]
//     Term 1 (AT2002-0250)/Term 2 (AT2002-5250)/FB Inputs/Value Channel 10 <-> Data Pointer/RawPositionValues[9]
//     Term 1 (AT2002-0250)/Term 2 (AT2002-5250)/FB Inputs/Value Channel 11 <-> Data Pointer/RawPositionValues[10]
//     Term 1 (AT2002-0250)/Term 2 (AT2002-5250)/FB Inputs/Value Channel 12 <-> Data Pointer/RawPositionValues[11]
//     Term 1 (AT2002-0250)/Term 2 (AT2002-5250)/FB Inputs/Value Channel 13 <-> Data Pointer/RawPositionValues[12]
//     Term 1 (AT2002-0250)/Term 2 (AT2002-5250)/FB Inputs/Value Channel 14 <-> Data Pointer/RawPositionValues[13]
//     Term 1 (AT2002-0250)/Term 2 (AT2002-5250)/FB Inputs/Value Channel 15 <-> Data Pointer/RawPositionValues[14]
//     Term 1 (AT2002-0250)/Term 2 (AT2002-5250)/FB Inputs/Value Channel 16 <-> Data Pointer/RawPositionValues[15]
//     Term 1 (AT2002-0250)/Term 2 (AT2002-5250)/FB Inputs/Value Channel 17 <-> Data Pointer/RawPositionValues[16]
//     Term 1 (AT2002-0250)/Term 2 (AT2002-5250)/FB Inputs/Value Channel 18 <-> Data Pointer/RawPositionValues[17]
//     Term 1 (AT2002-0250)/Term 2 (AT2002-5250)/FB Inputs/Value Channel 19 <-> Data Pointer/RawPositionValues[18]
//     Term 1 (AT2002-0250)/Term 2 (AT2002-5250)/FB Inputs/Value Channel 20 <-> Data Pointer/RawPositionValues[19]
//     Term 1 (AT2002-0250)/Term 2 (AT2002-5250)/FB Inputs/Value Channel 21 <-> Data Pointer/RawPositionValues[20]
//     Term 1 (AT2002-0250)/Term 2 (AT2002-5250)/FB Inputs/Value Channel 22 <-> Data Pointer/RawPositionValues[21]
//     Term 1 (AT2002-0250)/Term 2 (AT2002-5250)/FB Inputs/Value Channel 23 <-> Data Pointer/RawPositionValues[22]
//     Term 1 (AT2002-0250)/Term 2 (AT2002-5250)/FB Inputs/Value Channel 24 <-> Data Pointer/RawPositionValues[23]
//     Term 1 (AT2002-0250)/Term 2 (AT2002-5250)/FB Inputs/Value Channel 25 <-> Data Pointer/RawPositionValues[24]
//     Term 1 (AT2002-0250)/Term 2 (AT2002-5250)/FB Inputs/Value Channel 26 <-> Data Pointer/RawPositionValues[25]
//     Term 1 (AT2002-0250)/Term 2 (AT2002-5250)/FB Inputs/Value Channel 27 <-> Data Pointer/RawPositionValues[26]
//     Term 1 (AT2002-0250)/Term 2 (AT2002-5250)/FB Inputs/Value Channel 28 <-> Data Pointer/RawPositionValues[27]
//     Term 1 (AT2002-0250)/Term 2 (AT2002-5250)/FB Inputs/Value Channel 29 <-> Data Pointer/RawPositionValues[28]
//     Term 1 (AT2002-0250)/Term 2 (AT2002-5250)/FB Inputs/Value Channel 30 <-> Data Pointer/RawPositionValues[29]
//     Term 1 (AT2002-0250)/Term 2 (AT2002-5250)/FB Inputs/Value Channel 31 <-> Data Pointer/RawPositionValues[30]
//     Term 1 (AT2002-0250)/Term 2 (AT2002-5250)/FB Inputs/Value Channel 32 <-> Data Pointer/RawPositionValues[31]
//   Device 1 <-> TcCOM Objects/XTS ProcessingUnit 1/Part 1/Module 2
//     Term 3 (AT2000-0250)/CC Inputs/Current actual value Ch.1 <-> Data Pointer/CurrentActualValues[0]
//     Term 3 (AT2000-0250)/CC Inputs/Current actual value Ch.10 <-> Data Pointer/CurrentActualValues[9]
//     Term 3 (AT2000-0250)/CC Inputs/Current actual value Ch.11 <-> Data Pointer/CurrentActualValues[10]
//     Term 3 (AT2000-0250)/CC Inputs/Current actual value Ch.12 <-> Data Pointer/CurrentActualValues[11]
//     Term 3 (AT2000-0250)/CC Inputs/Current actual value Ch.13 <-> Data Pointer/CurrentActualValues[12]
//     Term 3 (AT2000-0250)/CC Inputs/Current actual value Ch.14 <-> Data Pointer/CurrentActualValues[13]
//     Term 3 (AT2000-0250)/CC Inputs/Current actual value Ch.15 <-> Data Pointer/CurrentActualValues[14]
//     Term 3 (AT2000-0250)/CC Inputs/Current actual value Ch.2 <-> Data Pointer/CurrentActualValues[1]
//     Term 3 (AT2000-0250)/CC Inputs/Current actual value Ch.3 <-> Data Pointer/CurrentActualValues[2]
//     Term 3 (AT2000-0250)/CC Inputs/Current actual value Ch.4 <-> Data Pointer/CurrentActualValues[3]
//     Term 3 (AT2000-0250)/CC Inputs/Current actual value Ch.5 <-> Data Pointer/CurrentActualValues[4]
//     Term 3 (AT2000-0250)/CC Inputs/Current actual value Ch.6 <-> Data Pointer/CurrentActualValues[5]
//     Term 3 (AT2000-0250)/CC Inputs/Current actual value Ch.7 <-> Data Pointer/CurrentActualValues[6]
//     Term 3 (AT2000-0250)/CC Inputs/Current actual value Ch.8 <-> Data Pointer/CurrentActualValues[7]
//     Term 3 (AT2000-0250)/CC Inputs/Current actual value Ch.9 <-> Data Pointer/CurrentActualValues[8]
//     Term 3 (AT2000-0250)/CC Inputs/Status <-> Data Pointer/Status
//     Term 3 (AT2000-0250)/CC Outputs/Control <-> Data Pointer/Control
//     Term 3 (AT2000-0250)/CC Outputs/Current setpoint value Ch.1 <-> Data Pointer/CurrentSetpointValues[0]
//     Term 3 (AT2000-0250)/CC Outputs/Current setpoint value Ch.10 <-> Data Pointer/CurrentSetpointValues[9]
//     Term 3 (AT2000-0250)/CC Outputs/Current setpoint value Ch.11 <-> Data Pointer/CurrentSetpointValues[10]
//     Term 3 (AT2000-0250)/CC Outputs/Current setpoint value Ch.12 <-> Data Pointer/CurrentSetpointValues[11]
//     Term 3 (AT2000-0250)/CC Outputs/Current setpoint value Ch.13 <-> Data Pointer/CurrentSetpointValues[12]
//     Term 3 (AT2000-0250)/CC Outputs/Current setpoint value Ch.14 <-> Data Pointer/CurrentSetpointValues[13]
//     Term 3 (AT2000-0250)/CC Outputs/Current setpoint value Ch.15 <-> Data Pointer/CurrentSetpointValues[14]
//     Term 3 (AT2000-0250)/CC Outputs/Current setpoint value Ch.2 <-> Data Pointer/CurrentSetpointValues[1]
//     Term 3 (AT2000-0250)/CC Outputs/Current setpoint value Ch.3 <-> Data Pointer/CurrentSetpointValues[2]
//     Term 3 (AT2000-0250)/CC Outputs/Current setpoint value Ch.4 <-> Data Pointer/CurrentSetpointValues[3]
//     Term 3 (AT2000-0250)/CC Outputs/Current setpoint value Ch.5 <-> Data Pointer/CurrentSetpointValues[4]
//     Term 3 (AT2000-0250)/CC Outputs/Current setpoint value Ch.6 <-> Data Pointer/CurrentSetpointValues[5]
//     Term 3 (AT2000-0250)/CC Outputs/Current setpoint value Ch.7 <-> Data Pointer/CurrentSetpointValues[6]
//     Term 3 (AT2000-0250)/CC Outputs/Current setpoint value Ch.8 <-> Data Pointer/CurrentSetpointValues[7]
//     Term 3 (AT2000-0250)/CC Outputs/Current setpoint value Ch.9 <-> Data Pointer/CurrentSetpointValues[8]
//     Term 3 (AT2000-0250)/Term 4 (AT2000-5250)/FB Inputs/Value Channel 01 <-> Data Pointer/RawPositionValues[0]
//     Term 3 (AT2000-0250)/Term 4 (AT2000-5250)/FB Inputs/Value Channel 02 <-> Data Pointer/RawPositionValues[1]
//     Term 3 (AT2000-0250)/Term 4 (AT2000-5250)/FB Inputs/Value Channel 03 <-> Data Pointer/RawPositionValues[2]
//     Term 3 (AT2000-0250)/Term 4 (AT2000-5250)/FB Inputs/Value Channel 04 <-> Data Pointer/RawPositionValues[3]
//     Term 3 (AT2000-0250)/Term 4 (AT2000-5250)/FB Inputs/Value Channel 05 <-> Data Pointer/RawPositionValues[4]
//     Term 3 (AT2000-0250)/Term 4 (AT2000-5250)/FB Inputs/Value Channel 06 <-> Data Pointer/RawPositionValues[5]
//     Term 3 (AT2000-0250)/Term 4 (AT2000-5250)/FB Inputs/Value Channel 07 <-> Data Pointer/RawPositionValues[6]
//     Term 3 (AT2000-0250)/Term 4 (AT2000-5250)/FB Inputs/Value Channel 08 <-> Data Pointer/RawPositionValues[7]
//     Term 3 (AT2000-0250)/Term 4 (AT2000-5250)/FB Inputs/Value Channel 09 <-> Data Pointer/RawPositionValues[8]
//     Term 3 (AT2000-0250)/Term 4 (AT2000-5250)/FB Inputs/Value Channel 10 <-> Data Pointer/RawPositionValues[9]
//     Term 3 (AT2000-0250)/Term 4 (AT2000-5250)/FB Inputs/Value Channel 11 <-> Data Pointer/RawPositionValues[10]
//     Term 3 (AT2000-0250)/Term 4 (AT2000-5250)/FB Inputs/Value Channel 12 <-> Data Pointer/RawPositionValues[11]
//     Term 3 (AT2000-0250)/Term 4 (AT2000-5250)/FB Inputs/Value Channel 13 <-> Data Pointer/RawPositionValues[12]
//     Term 3 (AT2000-0250)/Term 4 (AT2000-5250)/FB Inputs/Value Channel 14 <-> Data Pointer/RawPositionValues[13]
//     Term 3 (AT2000-0250)/Term 4 (AT2000-5250)/FB Inputs/Value Channel 15 <-> Data Pointer/RawPositionValues[14]
//     Term 3 (AT2000-0250)/Term 4 (AT2000-5250)/FB Inputs/Value Channel 16 <-> Data Pointer/RawPositionValues[15]
//     Term 3 (AT2000-0250)/Term 4 (AT2000-5250)/FB Inputs/Value Channel 17 <-> Data Pointer/RawPositionValues[16]
//     Term 3 (AT2000-0250)/Term 4 (AT2000-5250)/FB Inputs/Value Channel 18 <-> Data Pointer/RawPositionValues[17]
//     Term 3 (AT2000-0250)/Term 4 (AT2000-5250)/FB Inputs/Value Channel 19 <-> Data Pointer/RawPositionValues[18]
//     Term 3 (AT2000-0250)/Term 4 (AT2000-5250)/FB Inputs/Value Channel 20 <-> Data Pointer/RawPositionValues[19]
//     Term 3 (AT2000-0250)/Term 4 (AT2000-5250)/FB Inputs/Value Channel 21 <-> Data Pointer/RawPositionValues[20]
//     Term 3 (AT2000-0250)/Term 4 (AT2000-5250)/FB Inputs/Value Channel 22 <-> Data Pointer/RawPositionValues[21]
//     Term 3 (AT2000-0250)/Term 4 (AT2000-5250)/FB Inputs/Value Channel 23 <-> Data Pointer/RawPositionValues[22]
//     Term 3 (AT2000-0250)/Term 4 (AT2000-5250)/FB Inputs/Value Channel 24 <-> Data Pointer/RawPositionValues[23]
//     Term 3 (AT2000-0250)/Term 4 (AT2000-5250)/FB Inputs/Value Channel 25 <-> Data Pointer/RawPositionValues[24]
//     Term 3 (AT2000-0250)/Term 4 (AT2000-5250)/FB Inputs/Value Channel 26 <-> Data Pointer/RawPositionValues[25]
//     Term 3 (AT2000-0250)/Term 4 (AT2000-5250)/FB Inputs/Value Channel 27 <-> Data Pointer/RawPositionValues[26]
//     Term 3 (AT2000-0250)/Term 4 (AT2000-5250)/FB Inputs/Value Channel 28 <-> Data Pointer/RawPositionValues[27]
//     Term 3 (AT2000-0250)/Term 4 (AT2000-5250)/FB Inputs/Value Channel 29 <-> Data Pointer/RawPositionValues[28]
//     Term 3 (AT2000-0250)/Term 4 (AT2000-5250)/FB Inputs/Value Channel 30 <-> Data Pointer/RawPositionValues[29]
//     Term 3 (AT2000-0250)/Term 4 (AT2000-5250)/FB Inputs/Value Channel 31 <-> Data Pointer/RawPositionValues[30]
//     Term 3 (AT2000-0250)/Term 4 (AT2000-5250)/FB Inputs/Value Channel 32 <-> Data Pointer/RawPositionValues[31]
//   Device 1 <-> TcCOM Objects/XTS ProcessingUnit 1/Part 1/Module 3
//     Term 5 (AT2000-0250)/CC Inputs/Current actual value Ch.1 <-> Data Pointer/CurrentActualValues[0]
//     Term 5 (AT2000-0250)/CC Inputs/Current actual value Ch.10 <-> Data Pointer/CurrentActualValues[9]
//     Term 5 (AT2000-0250)/CC Inputs/Current actual value Ch.11 <-> Data Pointer/CurrentActualValues[10]
//     Term 5 (AT2000-0250)/CC Inputs/Current actual value Ch.12 <-> Data Pointer/CurrentActualValues[11]
//     Term 5 (AT2000-0250)/CC Inputs/Current actual value Ch.13 <-> Data Pointer/CurrentActualValues[12]
//     Term 5 (AT2000-0250)/CC Inputs/Current actual value Ch.14 <-> Data Pointer/CurrentActualValues[13]
//     Term 5 (AT2000-0250)/CC Inputs/Current actual value Ch.15 <-> Data Pointer/CurrentActualValues[14]
//     Term 5 (AT2000-0250)/CC Inputs/Current actual value Ch.2 <-> Data Pointer/CurrentActualValues[1]
//     Term 5 (AT2000-0250)/CC Inputs/Current actual value Ch.3 <-> Data Pointer/CurrentActualValues[2]
//     Term 5 (AT2000-0250)/CC Inputs/Current actual value Ch.4 <-> Data Pointer/CurrentActualValues[3]
//     Term 5 (AT2000-0250)/CC Inputs/Current actual value Ch.5 <-> Data Pointer/CurrentActualValues[4]
//     Term 5 (AT2000-0250)/CC Inputs/Current actual value Ch.6 <-> Data Pointer/CurrentActualValues[5]
//     Term 5 (AT2000-0250)/CC Inputs/Current actual value Ch.7 <-> Data Pointer/CurrentActualValues[6]
//     Term 5 (AT2000-0250)/CC Inputs/Current actual value Ch.8 <-> Data Pointer/CurrentActualValues[7]
//     Term 5 (AT2000-0250)/CC Inputs/Current actual value Ch.9 <-> Data Pointer/CurrentActualValues[8]
//     Term 5 (AT2000-0250)/CC Inputs/Status <-> Data Pointer/Status
//     Term 5 (AT2000-0250)/CC Outputs/Control <-> Data Pointer/Control
//     Term 5 (AT2000-0250)/CC Outputs/Current setpoint value Ch.1 <-> Data Pointer/CurrentSetpointValues[0]
//     Term 5 (AT2000-0250)/CC Outputs/Current setpoint value Ch.10 <-> Data Pointer/CurrentSetpointValues[9]
//     Term 5 (AT2000-0250)/CC Outputs/Current setpoint value Ch.11 <-> Data Pointer/CurrentSetpointValues[10]
//     Term 5 (AT2000-0250)/CC Outputs/Current setpoint value Ch.12 <-> Data Pointer/CurrentSetpointValues[11]
//     Term 5 (AT2000-0250)/CC Outputs/Current setpoint value Ch.13 <-> Data Pointer/CurrentSetpointValues[12]
//     Term 5 (AT2000-0250)/CC Outputs/Current setpoint value Ch.14 <-> Data Pointer/CurrentSetpointValues[13]
//     Term 5 (AT2000-0250)/CC Outputs/Current setpoint value Ch.15 <-> Data Pointer/CurrentSetpointValues[14]
//     Term 5 (AT2000-0250)/CC Outputs/Current setpoint value Ch.2 <-> Data Pointer/CurrentSetpointValues[1]
//     Term 5 (AT2000-0250)/CC Outputs/Current setpoint value Ch.3 <-> Data Pointer/CurrentSetpointValues[2]
//     Term 5 (AT2000-0250)/CC Outputs/Current setpoint value Ch.4 <-> Data Pointer/CurrentSetpointValues[3]
//     Term 5 (AT2000-0250)/CC Outputs/Current setpoint value Ch.5 <-> Data Pointer/CurrentSetpointValues[4]
//     Term 5 (AT2000-0250)/CC Outputs/Current setpoint value Ch.6 <-> Data Pointer/CurrentSetpointValues[5]
//     Term 5 (AT2000-0250)/CC Outputs/Current setpoint value Ch.7 <-> Data Pointer/CurrentSetpointValues[6]
//     Term 5 (AT2000-0250)/CC Outputs/Current setpoint value Ch.8 <-> Data Pointer/CurrentSetpointValues[7]
//     Term 5 (AT2000-0250)/CC Outputs/Current setpoint value Ch.9 <-> Data Pointer/CurrentSetpointValues[8]
//     Term 5 (AT2000-0250)/Term 6 (AT2000-5250)/FB Inputs/Value Channel 01 <-> Data Pointer/RawPositionValues[0]
//     Term 5 (AT2000-0250)/Term 6 (AT2000-5250)/FB Inputs/Value Channel 02 <-> Data Pointer/RawPositionValues[1]
//     Term 5 (AT2000-0250)/Term 6 (AT2000-5250)/FB Inputs/Value Channel 03 <-> Data Pointer/RawPositionValues[2]
//     Term 5 (AT2000-0250)/Term 6 (AT2000-5250)/FB Inputs/Value Channel 04 <-> Data Pointer/RawPositionValues[3]
//     Term 5 (AT2000-0250)/Term 6 (AT2000-5250)/FB Inputs/Value Channel 05 <-> Data Pointer/RawPositionValues[4]
//     Term 5 (AT2000-0250)/Term 6 (AT2000-5250)/FB Inputs/Value Channel 06 <-> Data Pointer/RawPositionValues[5]
//     Term 5 (AT2000-0250)/Term 6 (AT2000-5250)/FB Inputs/Value Channel 07 <-> Data Pointer/RawPositionValues[6]
//     Term 5 (AT2000-0250)/Term 6 (AT2000-5250)/FB Inputs/Value Channel 08 <-> Data Pointer/RawPositionValues[7]
//     Term 5 (AT2000-0250)/Term 6 (AT2000-5250)/FB Inputs/Value Channel 09 <-> Data Pointer/RawPositionValues[8]
//     Term 5 (AT2000-0250)/Term 6 (AT2000-5250)/FB Inputs/Value Channel 10 <-> Data Pointer/RawPositionValues[9]
//     Term 5 (AT2000-0250)/Term 6 (AT2000-5250)/FB Inputs/Value Channel 11 <-> Data Pointer/RawPositionValues[10]
//     Term 5 (AT2000-0250)/Term 6 (AT2000-5250)/FB Inputs/Value Channel 12 <-> Data Pointer/RawPositionValues[11]
//     Term 5 (AT2000-0250)/Term 6 (AT2000-5250)/FB Inputs/Value Channel 13 <-> Data Pointer/RawPositionValues[12]
//     Term 5 (AT2000-0250)/Term 6 (AT2000-5250)/FB Inputs/Value Channel 14 <-> Data Pointer/RawPositionValues[13]
//     Term 5 (AT2000-0250)/Term 6 (AT2000-5250)/FB Inputs/Value Channel 15 <-> Data Pointer/RawPositionValues[14]
//     Term 5 (AT2000-0250)/Term 6 (AT2000-5250)/FB Inputs/Value Channel 16 <-> Data Pointer/RawPositionValues[15]
//     Term 5 (AT2000-0250)/Term 6 (AT2000-5250)/FB Inputs/Value Channel 17 <-> Data Pointer/RawPositionValues[16]
//     Term 5 (AT2000-0250)/Term 6 (AT2000-5250)/FB Inputs/Value Channel 18 <-> Data Pointer/RawPositionValues[17]
//     Term 5 (AT2000-0250)/Term 6 (AT2000-5250)/FB Inputs/Value Channel 19 <-> Data Pointer/RawPositionValues[18]
//     Term 5 (AT2000-0250)/Term 6 (AT2000-5250)/FB Inputs/Value Channel 20 <-> Data Pointer/RawPositionValues[19]
//     Term 5 (AT2000-0250)/Term 6 (AT2000-5250)/FB Inputs/Value Channel 21 <-> Data Pointer/RawPositionValues[20]
//     Term 5 (AT2000-0250)/Term 6 (AT2000-5250)/FB Inputs/Value Channel 22 <-> Data Pointer/RawPositionValues[21]
//     Term 5 (AT2000-0250)/Term 6 (AT2000-5250)/FB Inputs/Value Channel 23 <-> Data Pointer/RawPositionValues[22]
//     Term 5 (AT2000-0250)/Term 6 (AT2000-5250)/FB Inputs/Value Channel 24 <-> Data Pointer/RawPositionValues[23]
//     Term 5 (AT2000-0250)/Term 6 (AT2000-5250)/FB Inputs/Value Channel 25 <-> Data Pointer/RawPositionValues[24]
//     Term 5 (AT2000-0250)/Term 6 (AT2000-5250)/FB Inputs/Value Channel 26 <-> Data Pointer/RawPositionValues[25]
//     Term 5 (AT2000-0250)/Term 6 (AT2000-5250)/FB Inputs/Value Channel 27 <-> Data Pointer/RawPositionValues[26]
//     Term 5 (AT2000-0250)/Term 6 (AT2000-5250)/FB Inputs/Value Channel 28 <-> Data Pointer/RawPositionValues[27]
//     Term 5 (AT2000-0250)/Term 6 (AT2000-5250)/FB Inputs/Value Channel 29 <-> Data Pointer/RawPositionValues[28]
//     Term 5 (AT2000-0250)/Term 6 (AT2000-5250)/FB Inputs/Value Channel 30 <-> Data Pointer/RawPositionValues[29]
//     Term 5 (AT2000-0250)/Term 6 (AT2000-5250)/FB Inputs/Value Channel 31 <-> Data Pointer/RawPositionValues[30]
//     Term 5 (AT2000-0250)/Term 6 (AT2000-5250)/FB Inputs/Value Channel 32 <-> Data Pointer/RawPositionValues[31]
//   Device 1 <-> TcCOM Objects/XTS ProcessingUnit 1/Part 1/Module 4
//     Term 7 (AT2000-0250)/CC Inputs/Current actual value Ch.1 <-> Data Pointer/CurrentActualValues[0]
//     Term 7 (AT2000-0250)/CC Inputs/Current actual value Ch.10 <-> Data Pointer/CurrentActualValues[9]
//     Term 7 (AT2000-0250)/CC Inputs/Current actual value Ch.11 <-> Data Pointer/CurrentActualValues[10]
//     Term 7 (AT2000-0250)/CC Inputs/Current actual value Ch.12 <-> Data Pointer/CurrentActualValues[11]
//     Term 7 (AT2000-0250)/CC Inputs/Current actual value Ch.13 <-> Data Pointer/CurrentActualValues[12]
//     Term 7 (AT2000-0250)/CC Inputs/Current actual value Ch.14 <-> Data Pointer/CurrentActualValues[13]
//     Term 7 (AT2000-0250)/CC Inputs/Current actual value Ch.15 <-> Data Pointer/CurrentActualValues[14]
//     Term 7 (AT2000-0250)/CC Inputs/Current actual value Ch.2 <-> Data Pointer/CurrentActualValues[1]
//     Term 7 (AT2000-0250)/CC Inputs/Current actual value Ch.3 <-> Data Pointer/CurrentActualValues[2]
//     Term 7 (AT2000-0250)/CC Inputs/Current actual value Ch.4 <-> Data Pointer/CurrentActualValues[3]
//     Term 7 (AT2000-0250)/CC Inputs/Current actual value Ch.5 <-> Data Pointer/CurrentActualValues[4]
//     Term 7 (AT2000-0250)/CC Inputs/Current actual value Ch.6 <-> Data Pointer/CurrentActualValues[5]
//     Term 7 (AT2000-0250)/CC Inputs/Current actual value Ch.7 <-> Data Pointer/CurrentActualValues[6]
//     Term 7 (AT2000-0250)/CC Inputs/Current actual value Ch.8 <-> Data Pointer/CurrentActualValues[7]
//     Term 7 (AT2000-0250)/CC Inputs/Current actual value Ch.9 <-> Data Pointer/CurrentActualValues[8]
//     Term 7 (AT2000-0250)/CC Inputs/Status <-> Data Pointer/Status
//     Term 7 (AT2000-0250)/CC Outputs/Control <-> Data Pointer/Control
//     Term 7 (AT2000-0250)/CC Outputs/Current setpoint value Ch.1 <-> Data Pointer/CurrentSetpointValues[0]
//     Term 7 (AT2000-0250)/CC Outputs/Current setpoint value Ch.10 <-> Data Pointer/CurrentSetpointValues[9]
//     Term 7 (AT2000-0250)/CC Outputs/Current setpoint value Ch.11 <-> Data Pointer/CurrentSetpointValues[10]
//     Term 7 (AT2000-0250)/CC Outputs/Current setpoint value Ch.12 <-> Data Pointer/CurrentSetpointValues[11]
//     Term 7 (AT2000-0250)/CC Outputs/Current setpoint value Ch.13 <-> Data Pointer/CurrentSetpointValues[12]
//     Term 7 (AT2000-0250)/CC Outputs/Current setpoint value Ch.14 <-> Data Pointer/CurrentSetpointValues[13]
//     Term 7 (AT2000-0250)/CC Outputs/Current setpoint value Ch.15 <-> Data Pointer/CurrentSetpointValues[14]
//     Term 7 (AT2000-0250)/CC Outputs/Current setpoint value Ch.2 <-> Data Pointer/CurrentSetpointValues[1]
//     Term 7 (AT2000-0250)/CC Outputs/Current setpoint value Ch.3 <-> Data Pointer/CurrentSetpointValues[2]
//     Term 7 (AT2000-0250)/CC Outputs/Current setpoint value Ch.4 <-> Data Pointer/CurrentSetpointValues[3]
//     Term 7 (AT2000-0250)/CC Outputs/Current setpoint value Ch.5 <-> Data Pointer/CurrentSetpointValues[4]
//     Term 7 (AT2000-0250)/CC Outputs/Current setpoint value Ch.6 <-> Data Pointer/CurrentSetpointValues[5]
//     Term 7 (AT2000-0250)/CC Outputs/Current setpoint value Ch.7 <-> Data Pointer/CurrentSetpointValues[6]
//     Term 7 (AT2000-0250)/CC Outputs/Current setpoint value Ch.8 <-> Data Pointer/CurrentSetpointValues[7]
//     Term 7 (AT2000-0250)/CC Outputs/Current setpoint value Ch.9 <-> Data Pointer/CurrentSetpointValues[8]
//     Term 7 (AT2000-0250)/Term 8 (AT2000-5250)/FB Inputs/Value Channel 01 <-> Data Pointer/RawPositionValues[0]
//     Term 7 (AT2000-0250)/Term 8 (AT2000-5250)/FB Inputs/Value Channel 02 <-> Data Pointer/RawPositionValues[1]
//     Term 7 (AT2000-0250)/Term 8 (AT2000-5250)/FB Inputs/Value Channel 03 <-> Data Pointer/RawPositionValues[2]
//     Term 7 (AT2000-0250)/Term 8 (AT2000-5250)/FB Inputs/Value Channel 04 <-> Data Pointer/RawPositionValues[3]
//     Term 7 (AT2000-0250)/Term 8 (AT2000-5250)/FB Inputs/Value Channel 05 <-> Data Pointer/RawPositionValues[4]
//     Term 7 (AT2000-0250)/Term 8 (AT2000-5250)/FB Inputs/Value Channel 06 <-> Data Pointer/RawPositionValues[5]
//     Term 7 (AT2000-0250)/Term 8 (AT2000-5250)/FB Inputs/Value Channel 07 <-> Data Pointer/RawPositionValues[6]
//     Term 7 (AT2000-0250)/Term 8 (AT2000-5250)/FB Inputs/Value Channel 08 <-> Data Pointer/RawPositionValues[7]
//     Term 7 (AT2000-0250)/Term 8 (AT2000-5250)/FB Inputs/Value Channel 09 <-> Data Pointer/RawPositionValues[8]
//     Term 7 (AT2000-0250)/Term 8 (AT2000-5250)/FB Inputs/Value Channel 10 <-> Data Pointer/RawPositionValues[9]
//     Term 7 (AT2000-0250)/Term 8 (AT2000-5250)/FB Inputs/Value Channel 11 <-> Data Pointer/RawPositionValues[10]
//     Term 7 (AT2000-0250)/Term 8 (AT2000-5250)/FB Inputs/Value Channel 12 <-> Data Pointer/RawPositionValues[11]
//     Term 7 (AT2000-0250)/Term 8 (AT2000-5250)/FB Inputs/Value Channel 13 <-> Data Pointer/RawPositionValues[12]
//     Term 7 (AT2000-0250)/Term 8 (AT2000-5250)/FB Inputs/Value Channel 14 <-> Data Pointer/RawPositionValues[13]
//     Term 7 (AT2000-0250)/Term 8 (AT2000-5250)/FB Inputs/Value Channel 15 <-> Data Pointer/RawPositionValues[14]
//     Term 7 (AT2000-0250)/Term 8 (AT2000-5250)/FB Inputs/Value Channel 16 <-> Data Pointer/RawPositionValues[15]
//     Term 7 (AT2000-0250)/Term 8 (AT2000-5250)/FB Inputs/Value Channel 17 <-> Data Pointer/RawPositionValues[16]
//     Term 7 (AT2000-0250)/Term 8 (AT2000-5250)/FB Inputs/Value Channel 18 <-> Data Pointer/RawPositionValues[17]
//     Term 7 (AT2000-0250)/Term 8 (AT2000-5250)/FB Inputs/Value Channel 19 <-> Data Pointer/RawPositionValues[18]
//     Term 7 (AT2000-0250)/Term 8 (AT2000-5250)/FB Inputs/Value Channel 20 <-> Data Pointer/RawPositionValues[19]
//     Term 7 (AT2000-0250)/Term 8 (AT2000-5250)/FB Inputs/Value Channel 21 <-> Data Pointer/RawPositionValues[20]
//     Term 7 (AT2000-0250)/Term 8 (AT2000-5250)/FB Inputs/Value Channel 22 <-> Data Pointer/RawPositionValues[21]
//     Term 7 (AT2000-0250)/Term 8 (AT2000-5250)/FB Inputs/Value Channel 23 <-> Data Pointer/RawPositionValues[22]
//     Term 7 (AT2000-0250)/Term 8 (AT2000-5250)/FB Inputs/Value Channel 24 <-> Data Pointer/RawPositionValues[23]
//     Term 7 (AT2000-0250)/Term 8 (AT2000-5250)/FB Inputs/Value Channel 25 <-> Data Pointer/RawPositionValues[24]
//     Term 7 (AT2000-0250)/Term 8 (AT2000-5250)/FB Inputs/Value Channel 26 <-> Data Pointer/RawPositionValues[25]
//     Term 7 (AT2000-0250)/Term 8 (AT2000-5250)/FB Inputs/Value Channel 27 <-> Data Pointer/RawPositionValues[26]
//     Term 7 (AT2000-0250)/Term 8 (AT2000-5250)/FB Inputs/Value Channel 28 <-> Data Pointer/RawPositionValues[27]
//     Term 7 (AT2000-0250)/Term 8 (AT2000-5250)/FB Inputs/Value Channel 29 <-> Data Pointer/RawPositionValues[28]
//     Term 7 (AT2000-0250)/Term 8 (AT2000-5250)/FB Inputs/Value Channel 30 <-> Data Pointer/RawPositionValues[29]
//     Term 7 (AT2000-0250)/Term 8 (AT2000-5250)/FB Inputs/Value Channel 31 <-> Data Pointer/RawPositionValues[30]
//     Term 7 (AT2000-0250)/Term 8 (AT2000-5250)/FB Inputs/Value Channel 32 <-> Data Pointer/RawPositionValues[31]
//   Device 3 <-> TcCOM Objects/XTS ProcessingUnit 1/Part 1/Module 5
//     Term 9 (AT2002-0250)/CC Inputs/Current actual value Ch.1 <-> Data Pointer/CurrentActualValues[0]
//     Term 9 (AT2002-0250)/CC Inputs/Current actual value Ch.10 <-> Data Pointer/CurrentActualValues[9]
//     Term 9 (AT2002-0250)/CC Inputs/Current actual value Ch.11 <-> Data Pointer/CurrentActualValues[10]
//     Term 9 (AT2002-0250)/CC Inputs/Current actual value Ch.12 <-> Data Pointer/CurrentActualValues[11]
//     Term 9 (AT2002-0250)/CC Inputs/Current actual value Ch.13 <-> Data Pointer/CurrentActualValues[12]
//     Term 9 (AT2002-0250)/CC Inputs/Current actual value Ch.14 <-> Data Pointer/CurrentActualValues[13]
//     Term 9 (AT2002-0250)/CC Inputs/Current actual value Ch.15 <-> Data Pointer/CurrentActualValues[14]
//     Term 9 (AT2002-0250)/CC Inputs/Current actual value Ch.2 <-> Data Pointer/CurrentActualValues[1]
//     Term 9 (AT2002-0250)/CC Inputs/Current actual value Ch.3 <-> Data Pointer/CurrentActualValues[2]
//     Term 9 (AT2002-0250)/CC Inputs/Current actual value Ch.4 <-> Data Pointer/CurrentActualValues[3]
//     Term 9 (AT2002-0250)/CC Inputs/Current actual value Ch.5 <-> Data Pointer/CurrentActualValues[4]
//     Term 9 (AT2002-0250)/CC Inputs/Current actual value Ch.6 <-> Data Pointer/CurrentActualValues[5]
//     Term 9 (AT2002-0250)/CC Inputs/Current actual value Ch.7 <-> Data Pointer/CurrentActualValues[6]
//     Term 9 (AT2002-0250)/CC Inputs/Current actual value Ch.8 <-> Data Pointer/CurrentActualValues[7]
//     Term 9 (AT2002-0250)/CC Inputs/Current actual value Ch.9 <-> Data Pointer/CurrentActualValues[8]
//     Term 9 (AT2002-0250)/CC Inputs/Status <-> Data Pointer/Status
//     Term 9 (AT2002-0250)/CC Outputs/Control <-> Data Pointer/Control
//     Term 9 (AT2002-0250)/CC Outputs/Current setpoint value Ch.1 <-> Data Pointer/CurrentSetpointValues[0]
//     Term 9 (AT2002-0250)/CC Outputs/Current setpoint value Ch.10 <-> Data Pointer/CurrentSetpointValues[9]
//     Term 9 (AT2002-0250)/CC Outputs/Current setpoint value Ch.11 <-> Data Pointer/CurrentSetpointValues[10]
//     Term 9 (AT2002-0250)/CC Outputs/Current setpoint value Ch.12 <-> Data Pointer/CurrentSetpointValues[11]
//     Term 9 (AT2002-0250)/CC Outputs/Current setpoint value Ch.13 <-> Data Pointer/CurrentSetpointValues[12]
//     Term 9 (AT2002-0250)/CC Outputs/Current setpoint value Ch.14 <-> Data Pointer/CurrentSetpointValues[13]
//     Term 9 (AT2002-0250)/CC Outputs/Current setpoint value Ch.15 <-> Data Pointer/CurrentSetpointValues[14]
//     Term 9 (AT2002-0250)/CC Outputs/Current setpoint value Ch.2 <-> Data Pointer/CurrentSetpointValues[1]
//     Term 9 (AT2002-0250)/CC Outputs/Current setpoint value Ch.3 <-> Data Pointer/CurrentSetpointValues[2]
//     Term 9 (AT2002-0250)/CC Outputs/Current setpoint value Ch.4 <-> Data Pointer/CurrentSetpointValues[3]
//     Term 9 (AT2002-0250)/CC Outputs/Current setpoint value Ch.5 <-> Data Pointer/CurrentSetpointValues[4]
//     Term 9 (AT2002-0250)/CC Outputs/Current setpoint value Ch.6 <-> Data Pointer/CurrentSetpointValues[5]
//     Term 9 (AT2002-0250)/CC Outputs/Current setpoint value Ch.7 <-> Data Pointer/CurrentSetpointValues[6]
//     Term 9 (AT2002-0250)/CC Outputs/Current setpoint value Ch.8 <-> Data Pointer/CurrentSetpointValues[7]
//     Term 9 (AT2002-0250)/CC Outputs/Current setpoint value Ch.9 <-> Data Pointer/CurrentSetpointValues[8]
//     Term 9 (AT2002-0250)/Term 10 (AT2002-5250)/FB Inputs/Value Channel 01 <-> Data Pointer/RawPositionValues[0]
//     Term 9 (AT2002-0250)/Term 10 (AT2002-5250)/FB Inputs/Value Channel 02 <-> Data Pointer/RawPositionValues[1]
//     Term 9 (AT2002-0250)/Term 10 (AT2002-5250)/FB Inputs/Value Channel 03 <-> Data Pointer/RawPositionValues[2]
//     Term 9 (AT2002-0250)/Term 10 (AT2002-5250)/FB Inputs/Value Channel 04 <-> Data Pointer/RawPositionValues[3]
//     Term 9 (AT2002-0250)/Term 10 (AT2002-5250)/FB Inputs/Value Channel 05 <-> Data Pointer/RawPositionValues[4]
//     Term 9 (AT2002-0250)/Term 10 (AT2002-5250)/FB Inputs/Value Channel 06 <-> Data Pointer/RawPositionValues[5]
//     Term 9 (AT2002-0250)/Term 10 (AT2002-5250)/FB Inputs/Value Channel 07 <-> Data Pointer/RawPositionValues[6]
//     Term 9 (AT2002-0250)/Term 10 (AT2002-5250)/FB Inputs/Value Channel 08 <-> Data Pointer/RawPositionValues[7]
//     Term 9 (AT2002-0250)/Term 10 (AT2002-5250)/FB Inputs/Value Channel 09 <-> Data Pointer/RawPositionValues[8]
//     Term 9 (AT2002-0250)/Term 10 (AT2002-5250)/FB Inputs/Value Channel 10 <-> Data Pointer/RawPositionValues[9]
//     Term 9 (AT2002-0250)/Term 10 (AT2002-5250)/FB Inputs/Value Channel 11 <-> Data Pointer/RawPositionValues[10]
//     Term 9 (AT2002-0250)/Term 10 (AT2002-5250)/FB Inputs/Value Channel 12 <-> Data Pointer/RawPositionValues[11]
//     Term 9 (AT2002-0250)/Term 10 (AT2002-5250)/FB Inputs/Value Channel 13 <-> Data Pointer/RawPositionValues[12]
//     Term 9 (AT2002-0250)/Term 10 (AT2002-5250)/FB Inputs/Value Channel 14 <-> Data Pointer/RawPositionValues[13]
//     Term 9 (AT2002-0250)/Term 10 (AT2002-5250)/FB Inputs/Value Channel 15 <-> Data Pointer/RawPositionValues[14]
//     Term 9 (AT2002-0250)/Term 10 (AT2002-5250)/FB Inputs/Value Channel 16 <-> Data Pointer/RawPositionValues[15]
//     Term 9 (AT2002-0250)/Term 10 (AT2002-5250)/FB Inputs/Value Channel 17 <-> Data Pointer/RawPositionValues[16]
//     Term 9 (AT2002-0250)/Term 10 (AT2002-5250)/FB Inputs/Value Channel 18 <-> Data Pointer/RawPositionValues[17]
//     Term 9 (AT2002-0250)/Term 10 (AT2002-5250)/FB Inputs/Value Channel 19 <-> Data Pointer/RawPositionValues[18]
//     Term 9 (AT2002-0250)/Term 10 (AT2002-5250)/FB Inputs/Value Channel 20 <-> Data Pointer/RawPositionValues[19]
//     Term 9 (AT2002-0250)/Term 10 (AT2002-5250)/FB Inputs/Value Channel 21 <-> Data Pointer/RawPositionValues[20]
//     Term 9 (AT2002-0250)/Term 10 (AT2002-5250)/FB Inputs/Value Channel 22 <-> Data Pointer/RawPositionValues[21]
//     Term 9 (AT2002-0250)/Term 10 (AT2002-5250)/FB Inputs/Value Channel 23 <-> Data Pointer/RawPositionValues[22]
//     Term 9 (AT2002-0250)/Term 10 (AT2002-5250)/FB Inputs/Value Channel 24 <-> Data Pointer/RawPositionValues[23]
//     Term 9 (AT2002-0250)/Term 10 (AT2002-5250)/FB Inputs/Value Channel 25 <-> Data Pointer/RawPositionValues[24]
//     Term 9 (AT2002-0250)/Term 10 (AT2002-5250)/FB Inputs/Value Channel 26 <-> Data Pointer/RawPositionValues[25]
//     Term 9 (AT2002-0250)/Term 10 (AT2002-5250)/FB Inputs/Value Channel 27 <-> Data Pointer/RawPositionValues[26]
//     Term 9 (AT2002-0250)/Term 10 (AT2002-5250)/FB Inputs/Value Channel 28 <-> Data Pointer/RawPositionValues[27]
//     Term 9 (AT2002-0250)/Term 10 (AT2002-5250)/FB Inputs/Value Channel 29 <-> Data Pointer/RawPositionValues[28]
//     Term 9 (AT2002-0250)/Term 10 (AT2002-5250)/FB Inputs/Value Channel 30 <-> Data Pointer/RawPositionValues[29]
//     Term 9 (AT2002-0250)/Term 10 (AT2002-5250)/FB Inputs/Value Channel 31 <-> Data Pointer/RawPositionValues[30]
//     Term 9 (AT2002-0250)/Term 10 (AT2002-5250)/FB Inputs/Value Channel 32 <-> Data Pointer/RawPositionValues[31]
//   Device 3 <-> TcCOM Objects/XTS ProcessingUnit 1/Part 1/Module 6
//     Term 11 (AT2000-0250)/CC Inputs/Current actual value Ch.1 <-> Data Pointer/CurrentActualValues[0]
//     Term 11 (AT2000-0250)/CC Inputs/Current actual value Ch.10 <-> Data Pointer/CurrentActualValues[9]
//     Term 11 (AT2000-0250)/CC Inputs/Current actual value Ch.11 <-> Data Pointer/CurrentActualValues[10]
//     Term 11 (AT2000-0250)/CC Inputs/Current actual value Ch.12 <-> Data Pointer/CurrentActualValues[11]
//     Term 11 (AT2000-0250)/CC Inputs/Current actual value Ch.13 <-> Data Pointer/CurrentActualValues[12]
//     Term 11 (AT2000-0250)/CC Inputs/Current actual value Ch.14 <-> Data Pointer/CurrentActualValues[13]
//     Term 11 (AT2000-0250)/CC Inputs/Current actual value Ch.15 <-> Data Pointer/CurrentActualValues[14]
//     Term 11 (AT2000-0250)/CC Inputs/Current actual value Ch.2 <-> Data Pointer/CurrentActualValues[1]
//     Term 11 (AT2000-0250)/CC Inputs/Current actual value Ch.3 <-> Data Pointer/CurrentActualValues[2]
//     Term 11 (AT2000-0250)/CC Inputs/Current actual value Ch.4 <-> Data Pointer/CurrentActualValues[3]
//     Term 11 (AT2000-0250)/CC Inputs/Current actual value Ch.5 <-> Data Pointer/CurrentActualValues[4]
//     Term 11 (AT2000-0250)/CC Inputs/Current actual value Ch.6 <-> Data Pointer/CurrentActualValues[5]
//     Term 11 (AT2000-0250)/CC Inputs/Current actual value Ch.7 <-> Data Pointer/CurrentActualValues[6]
//     Term 11 (AT2000-0250)/CC Inputs/Current actual value Ch.8 <-> Data Pointer/CurrentActualValues[7]
//     Term 11 (AT2000-0250)/CC Inputs/Current actual value Ch.9 <-> Data Pointer/CurrentActualValues[8]
//     Term 11 (AT2000-0250)/CC Inputs/Status <-> Data Pointer/Status
//     Term 11 (AT2000-0250)/CC Outputs/Control <-> Data Pointer/Control
//     Term 11 (AT2000-0250)/CC Outputs/Current setpoint value Ch.1 <-> Data Pointer/CurrentSetpointValues[0]
//     Term 11 (AT2000-0250)/CC Outputs/Current setpoint value Ch.10 <-> Data Pointer/CurrentSetpointValues[9]
//     Term 11 (AT2000-0250)/CC Outputs/Current setpoint value Ch.11 <-> Data Pointer/CurrentSetpointValues[10]
//     Term 11 (AT2000-0250)/CC Outputs/Current setpoint value Ch.12 <-> Data Pointer/CurrentSetpointValues[11]
//     Term 11 (AT2000-0250)/CC Outputs/Current setpoint value Ch.13 <-> Data Pointer/CurrentSetpointValues[12]
//     Term 11 (AT2000-0250)/CC Outputs/Current setpoint value Ch.14 <-> Data Pointer/CurrentSetpointValues[13]
//     Term 11 (AT2000-0250)/CC Outputs/Current setpoint value Ch.15 <-> Data Pointer/CurrentSetpointValues[14]
//     Term 11 (AT2000-0250)/CC Outputs/Current setpoint value Ch.2 <-> Data Pointer/CurrentSetpointValues[1]
//     Term 11 (AT2000-0250)/CC Outputs/Current setpoint value Ch.3 <-> Data Pointer/CurrentSetpointValues[2]
//     Term 11 (AT2000-0250)/CC Outputs/Current setpoint value Ch.4 <-> Data Pointer/CurrentSetpointValues[3]
//     Term 11 (AT2000-0250)/CC Outputs/Current setpoint value Ch.5 <-> Data Pointer/CurrentSetpointValues[4]
//     Term 11 (AT2000-0250)/CC Outputs/Current setpoint value Ch.6 <-> Data Pointer/CurrentSetpointValues[5]
//     Term 11 (AT2000-0250)/CC Outputs/Current setpoint value Ch.7 <-> Data Pointer/CurrentSetpointValues[6]
//     Term 11 (AT2000-0250)/CC Outputs/Current setpoint value Ch.8 <-> Data Pointer/CurrentSetpointValues[7]
//     Term 11 (AT2000-0250)/CC Outputs/Current setpoint value Ch.9 <-> Data Pointer/CurrentSetpointValues[8]
//     Term 11 (AT2000-0250)/Term 12 (AT2000-5250)/FB Inputs/Value Channel 01 <-> Data Pointer/RawPositionValues[0]
//     Term 11 (AT2000-0250)/Term 12 (AT2000-5250)/FB Inputs/Value Channel 02 <-> Data Pointer/RawPositionValues[1]
//     Term 11 (AT2000-0250)/Term 12 (AT2000-5250)/FB Inputs/Value Channel 03 <-> Data Pointer/RawPositionValues[2]
//     Term 11 (AT2000-0250)/Term 12 (AT2000-5250)/FB Inputs/Value Channel 04 <-> Data Pointer/RawPositionValues[3]
//     Term 11 (AT2000-0250)/Term 12 (AT2000-5250)/FB Inputs/Value Channel 05 <-> Data Pointer/RawPositionValues[4]
//     Term 11 (AT2000-0250)/Term 12 (AT2000-5250)/FB Inputs/Value Channel 06 <-> Data Pointer/RawPositionValues[5]
//     Term 11 (AT2000-0250)/Term 12 (AT2000-5250)/FB Inputs/Value Channel 07 <-> Data Pointer/RawPositionValues[6]
//     Term 11 (AT2000-0250)/Term 12 (AT2000-5250)/FB Inputs/Value Channel 08 <-> Data Pointer/RawPositionValues[7]
//     Term 11 (AT2000-0250)/Term 12 (AT2000-5250)/FB Inputs/Value Channel 09 <-> Data Pointer/RawPositionValues[8]
//     Term 11 (AT2000-0250)/Term 12 (AT2000-5250)/FB Inputs/Value Channel 10 <-> Data Pointer/RawPositionValues[9]
//     Term 11 (AT2000-0250)/Term 12 (AT2000-5250)/FB Inputs/Value Channel 11 <-> Data Pointer/RawPositionValues[10]
//     Term 11 (AT2000-0250)/Term 12 (AT2000-5250)/FB Inputs/Value Channel 12 <-> Data Pointer/RawPositionValues[11]
//     Term 11 (AT2000-0250)/Term 12 (AT2000-5250)/FB Inputs/Value Channel 13 <-> Data Pointer/RawPositionValues[12]
//     Term 11 (AT2000-0250)/Term 12 (AT2000-5250)/FB Inputs/Value Channel 14 <-> Data Pointer/RawPositionValues[13]
//     Term 11 (AT2000-0250)/Term 12 (AT2000-5250)/FB Inputs/Value Channel 15 <-> Data Pointer/RawPositionValues[14]
//     Term 11 (AT2000-0250)/Term 12 (AT2000-5250)/FB Inputs/Value Channel 16 <-> Data Pointer/RawPositionValues[15]
//     Term 11 (AT2000-0250)/Term 12 (AT2000-5250)/FB Inputs/Value Channel 17 <-> Data Pointer/RawPositionValues[16]
//     Term 11 (AT2000-0250)/Term 12 (AT2000-5250)/FB Inputs/Value Channel 18 <-> Data Pointer/RawPositionValues[17]
//     Term 11 (AT2000-0250)/Term 12 (AT2000-5250)/FB Inputs/Value Channel 19 <-> Data Pointer/RawPositionValues[18]
//     Term 11 (AT2000-0250)/Term 12 (AT2000-5250)/FB Inputs/Value Channel 20 <-> Data Pointer/RawPositionValues[19]
//     Term 11 (AT2000-0250)/Term 12 (AT2000-5250)/FB Inputs/Value Channel 21 <-> Data Pointer/RawPositionValues[20]
//     Term 11 (AT2000-0250)/Term 12 (AT2000-5250)/FB Inputs/Value Channel 22 <-> Data Pointer/RawPositionValues[21]
//     Term 11 (AT2000-0250)/Term 12 (AT2000-5250)/FB Inputs/Value Channel 23 <-> Data Pointer/RawPositionValues[22]
//     Term 11 (AT2000-0250)/Term 12 (AT2000-5250)/FB Inputs/Value Channel 24 <-> Data Pointer/RawPositionValues[23]
//     Term 11 (AT2000-0250)/Term 12 (AT2000-5250)/FB Inputs/Value Channel 25 <-> Data Pointer/RawPositionValues[24]
//     Term 11 (AT2000-0250)/Term 12 (AT2000-5250)/FB Inputs/Value Channel 26 <-> Data Pointer/RawPositionValues[25]
//     Term 11 (AT2000-0250)/Term 12 (AT2000-5250)/FB Inputs/Value Channel 27 <-> Data Pointer/RawPositionValues[26]
//     Term 11 (AT2000-0250)/Term 12 (AT2000-5250)/FB Inputs/Value Channel 28 <-> Data Pointer/RawPositionValues[27]
//     Term 11 (AT2000-0250)/Term 12 (AT2000-5250)/FB Inputs/Value Channel 29 <-> Data Pointer/RawPositionValues[28]
//     Term 11 (AT2000-0250)/Term 12 (AT2000-5250)/FB Inputs/Value Channel 30 <-> Data Pointer/RawPositionValues[29]
//     Term 11 (AT2000-0250)/Term 12 (AT2000-5250)/FB Inputs/Value Channel 31 <-> Data Pointer/RawPositionValues[30]
//     Term 11 (AT2000-0250)/Term 12 (AT2000-5250)/FB Inputs/Value Channel 32 <-> Data Pointer/RawPositionValues[31]
//   Device 3 <-> TcCOM Objects/XTS ProcessingUnit 1/Part 1/Module 7
//     Term 13 (AT2000-0250)/CC Inputs/Current actual value Ch.1 <-> Data Pointer/CurrentActualValues[0]
//     Term 13 (AT2000-0250)/CC Inputs/Current actual value Ch.10 <-> Data Pointer/CurrentActualValues[9]
//     Term 13 (AT2000-0250)/CC Inputs/Current actual value Ch.11 <-> Data Pointer/CurrentActualValues[10]
//     Term 13 (AT2000-0250)/CC Inputs/Current actual value Ch.12 <-> Data Pointer/CurrentActualValues[11]
//     Term 13 (AT2000-0250)/CC Inputs/Current actual value Ch.13 <-> Data Pointer/CurrentActualValues[12]
//     Term 13 (AT2000-0250)/CC Inputs/Current actual value Ch.14 <-> Data Pointer/CurrentActualValues[13]
//     Term 13 (AT2000-0250)/CC Inputs/Current actual value Ch.15 <-> Data Pointer/CurrentActualValues[14]
//     Term 13 (AT2000-0250)/CC Inputs/Current actual value Ch.2 <-> Data Pointer/CurrentActualValues[1]
//     Term 13 (AT2000-0250)/CC Inputs/Current actual value Ch.3 <-> Data Pointer/CurrentActualValues[2]
//     Term 13 (AT2000-0250)/CC Inputs/Current actual value Ch.4 <-> Data Pointer/CurrentActualValues[3]
//     Term 13 (AT2000-0250)/CC Inputs/Current actual value Ch.5 <-> Data Pointer/CurrentActualValues[4]
//     Term 13 (AT2000-0250)/CC Inputs/Current actual value Ch.6 <-> Data Pointer/CurrentActualValues[5]
//     Term 13 (AT2000-0250)/CC Inputs/Current actual value Ch.7 <-> Data Pointer/CurrentActualValues[6]
//     Term 13 (AT2000-0250)/CC Inputs/Current actual value Ch.8 <-> Data Pointer/CurrentActualValues[7]
//     Term 13 (AT2000-0250)/CC Inputs/Current actual value Ch.9 <-> Data Pointer/CurrentActualValues[8]
//     Term 13 (AT2000-0250)/CC Inputs/Status <-> Data Pointer/Status
//     Term 13 (AT2000-0250)/CC Outputs/Control <-> Data Pointer/Control
//     Term 13 (AT2000-0250)/CC Outputs/Current setpoint value Ch.1 <-> Data Pointer/CurrentSetpointValues[0]
//     Term 13 (AT2000-0250)/CC Outputs/Current setpoint value Ch.10 <-> Data Pointer/CurrentSetpointValues[9]
//     Term 13 (AT2000-0250)/CC Outputs/Current setpoint value Ch.11 <-> Data Pointer/CurrentSetpointValues[10]
//     Term 13 (AT2000-0250)/CC Outputs/Current setpoint value Ch.12 <-> Data Pointer/CurrentSetpointValues[11]
//     Term 13 (AT2000-0250)/CC Outputs/Current setpoint value Ch.13 <-> Data Pointer/CurrentSetpointValues[12]
//     Term 13 (AT2000-0250)/CC Outputs/Current setpoint value Ch.14 <-> Data Pointer/CurrentSetpointValues[13]
//     Term 13 (AT2000-0250)/CC Outputs/Current setpoint value Ch.15 <-> Data Pointer/CurrentSetpointValues[14]
//     Term 13 (AT2000-0250)/CC Outputs/Current setpoint value Ch.2 <-> Data Pointer/CurrentSetpointValues[1]
//     Term 13 (AT2000-0250)/CC Outputs/Current setpoint value Ch.3 <-> Data Pointer/CurrentSetpointValues[2]
//     Term 13 (AT2000-0250)/CC Outputs/Current setpoint value Ch.4 <-> Data Pointer/CurrentSetpointValues[3]
//     Term 13 (AT2000-0250)/CC Outputs/Current setpoint value Ch.5 <-> Data Pointer/CurrentSetpointValues[4]
//     Term 13 (AT2000-0250)/CC Outputs/Current setpoint value Ch.6 <-> Data Pointer/CurrentSetpointValues[5]
//     Term 13 (AT2000-0250)/CC Outputs/Current setpoint value Ch.7 <-> Data Pointer/CurrentSetpointValues[6]
//     Term 13 (AT2000-0250)/CC Outputs/Current setpoint value Ch.8 <-> Data Pointer/CurrentSetpointValues[7]
//     Term 13 (AT2000-0250)/CC Outputs/Current setpoint value Ch.9 <-> Data Pointer/CurrentSetpointValues[8]
//     Term 13 (AT2000-0250)/Term 14 (AT2000-5250)/FB Inputs/Value Channel 01 <-> Data Pointer/RawPositionValues[0]
//     Term 13 (AT2000-0250)/Term 14 (AT2000-5250)/FB Inputs/Value Channel 02 <-> Data Pointer/RawPositionValues[1]
//     Term 13 (AT2000-0250)/Term 14 (AT2000-5250)/FB Inputs/Value Channel 03 <-> Data Pointer/RawPositionValues[2]
//     Term 13 (AT2000-0250)/Term 14 (AT2000-5250)/FB Inputs/Value Channel 04 <-> Data Pointer/RawPositionValues[3]
//     Term 13 (AT2000-0250)/Term 14 (AT2000-5250)/FB Inputs/Value Channel 05 <-> Data Pointer/RawPositionValues[4]
//     Term 13 (AT2000-0250)/Term 14 (AT2000-5250)/FB Inputs/Value Channel 06 <-> Data Pointer/RawPositionValues[5]
//     Term 13 (AT2000-0250)/Term 14 (AT2000-5250)/FB Inputs/Value Channel 07 <-> Data Pointer/RawPositionValues[6]
//     Term 13 (AT2000-0250)/Term 14 (AT2000-5250)/FB Inputs/Value Channel 08 <-> Data Pointer/RawPositionValues[7]
//     Term 13 (AT2000-0250)/Term 14 (AT2000-5250)/FB Inputs/Value Channel 09 <-> Data Pointer/RawPositionValues[8]
//     Term 13 (AT2000-0250)/Term 14 (AT2000-5250)/FB Inputs/Value Channel 10 <-> Data Pointer/RawPositionValues[9]
//     Term 13 (AT2000-0250)/Term 14 (AT2000-5250)/FB Inputs/Value Channel 11 <-> Data Pointer/RawPositionValues[10]
//     Term 13 (AT2000-0250)/Term 14 (AT2000-5250)/FB Inputs/Value Channel 12 <-> Data Pointer/RawPositionValues[11]
//     Term 13 (AT2000-0250)/Term 14 (AT2000-5250)/FB Inputs/Value Channel 13 <-> Data Pointer/RawPositionValues[12]
//     Term 13 (AT2000-0250)/Term 14 (AT2000-5250)/FB Inputs/Value Channel 14 <-> Data Pointer/RawPositionValues[13]
//     Term 13 (AT2000-0250)/Term 14 (AT2000-5250)/FB Inputs/Value Channel 15 <-> Data Pointer/RawPositionValues[14]
//     Term 13 (AT2000-0250)/Term 14 (AT2000-5250)/FB Inputs/Value Channel 16 <-> Data Pointer/RawPositionValues[15]
//     Term 13 (AT2000-0250)/Term 14 (AT2000-5250)/FB Inputs/Value Channel 17 <-> Data Pointer/RawPositionValues[16]
//     Term 13 (AT2000-0250)/Term 14 (AT2000-5250)/FB Inputs/Value Channel 18 <-> Data Pointer/RawPositionValues[17]
//     Term 13 (AT2000-0250)/Term 14 (AT2000-5250)/FB Inputs/Value Channel 19 <-> Data Pointer/RawPositionValues[18]
//     Term 13 (AT2000-0250)/Term 14 (AT2000-5250)/FB Inputs/Value Channel 20 <-> Data Pointer/RawPositionValues[19]
//     Term 13 (AT2000-0250)/Term 14 (AT2000-5250)/FB Inputs/Value Channel 21 <-> Data Pointer/RawPositionValues[20]
//     Term 13 (AT2000-0250)/Term 14 (AT2000-5250)/FB Inputs/Value Channel 22 <-> Data Pointer/RawPositionValues[21]
//     Term 13 (AT2000-0250)/Term 14 (AT2000-5250)/FB Inputs/Value Channel 23 <-> Data Pointer/RawPositionValues[22]
//     Term 13 (AT2000-0250)/Term 14 (AT2000-5250)/FB Inputs/Value Channel 24 <-> Data Pointer/RawPositionValues[23]
//     Term 13 (AT2000-0250)/Term 14 (AT2000-5250)/FB Inputs/Value Channel 25 <-> Data Pointer/RawPositionValues[24]
//     Term 13 (AT2000-0250)/Term 14 (AT2000-5250)/FB Inputs/Value Channel 26 <-> Data Pointer/RawPositionValues[25]
//     Term 13 (AT2000-0250)/Term 14 (AT2000-5250)/FB Inputs/Value Channel 27 <-> Data Pointer/RawPositionValues[26]
//     Term 13 (AT2000-0250)/Term 14 (AT2000-5250)/FB Inputs/Value Channel 28 <-> Data Pointer/RawPositionValues[27]
//     Term 13 (AT2000-0250)/Term 14 (AT2000-5250)/FB Inputs/Value Channel 29 <-> Data Pointer/RawPositionValues[28]
//     Term 13 (AT2000-0250)/Term 14 (AT2000-5250)/FB Inputs/Value Channel 30 <-> Data Pointer/RawPositionValues[29]
//     Term 13 (AT2000-0250)/Term 14 (AT2000-5250)/FB Inputs/Value Channel 31 <-> Data Pointer/RawPositionValues[30]
//     Term 13 (AT2000-0250)/Term 14 (AT2000-5250)/FB Inputs/Value Channel 32 <-> Data Pointer/RawPositionValues[31]
//   Device 3 <-> TcCOM Objects/XTS ProcessingUnit 1/Part 1/Module 8
//     Term 15 (AT2000-0250)/CC Inputs/Current actual value Ch.1 <-> Data Pointer/CurrentActualValues[0]
//     Term 15 (AT2000-0250)/CC Inputs/Current actual value Ch.10 <-> Data Pointer/CurrentActualValues[9]
//     Term 15 (AT2000-0250)/CC Inputs/Current actual value Ch.11 <-> Data Pointer/CurrentActualValues[10]
//     Term 15 (AT2000-0250)/CC Inputs/Current actual value Ch.12 <-> Data Pointer/CurrentActualValues[11]
//     Term 15 (AT2000-0250)/CC Inputs/Current actual value Ch.13 <-> Data Pointer/CurrentActualValues[12]
//     Term 15 (AT2000-0250)/CC Inputs/Current actual value Ch.14 <-> Data Pointer/CurrentActualValues[13]
//     Term 15 (AT2000-0250)/CC Inputs/Current actual value Ch.15 <-> Data Pointer/CurrentActualValues[14]
//     Term 15 (AT2000-0250)/CC Inputs/Current actual value Ch.2 <-> Data Pointer/CurrentActualValues[1]
//     Term 15 (AT2000-0250)/CC Inputs/Current actual value Ch.3 <-> Data Pointer/CurrentActualValues[2]
//     Term 15 (AT2000-0250)/CC Inputs/Current actual value Ch.4 <-> Data Pointer/CurrentActualValues[3]
//     Term 15 (AT2000-0250)/CC Inputs/Current actual value Ch.5 <-> Data Pointer/CurrentActualValues[4]
//     Term 15 (AT2000-0250)/CC Inputs/Current actual value Ch.6 <-> Data Pointer/CurrentActualValues[5]
//     Term 15 (AT2000-0250)/CC Inputs/Current actual value Ch.7 <-> Data Pointer/CurrentActualValues[6]
//     Term 15 (AT2000-0250)/CC Inputs/Current actual value Ch.8 <-> Data Pointer/CurrentActualValues[7]
//     Term 15 (AT2000-0250)/CC Inputs/Current actual value Ch.9 <-> Data Pointer/CurrentActualValues[8]
//     Term 15 (AT2000-0250)/CC Inputs/Status <-> Data Pointer/Status
//     Term 15 (AT2000-0250)/CC Outputs/Control <-> Data Pointer/Control
//     Term 15 (AT2000-0250)/CC Outputs/Current setpoint value Ch.1 <-> Data Pointer/CurrentSetpointValues[0]
//     Term 15 (AT2000-0250)/CC Outputs/Current setpoint value Ch.10 <-> Data Pointer/CurrentSetpointValues[9]
//     Term 15 (AT2000-0250)/CC Outputs/Current setpoint value Ch.11 <-> Data Pointer/CurrentSetpointValues[10]
//     Term 15 (AT2000-0250)/CC Outputs/Current setpoint value Ch.12 <-> Data Pointer/CurrentSetpointValues[11]
//     Term 15 (AT2000-0250)/CC Outputs/Current setpoint value Ch.13 <-> Data Pointer/CurrentSetpointValues[12]
//     Term 15 (AT2000-0250)/CC Outputs/Current setpoint value Ch.14 <-> Data Pointer/CurrentSetpointValues[13]
//     Term 15 (AT2000-0250)/CC Outputs/Current setpoint value Ch.15 <-> Data Pointer/CurrentSetpointValues[14]
//     Term 15 (AT2000-0250)/CC Outputs/Current setpoint value Ch.2 <-> Data Pointer/CurrentSetpointValues[1]
//     Term 15 (AT2000-0250)/CC Outputs/Current setpoint value Ch.3 <-> Data Pointer/CurrentSetpointValues[2]
